REGION Network 4: First Cylinder No-3
   RUNG wire#powerrail
      Contact( "AlwaysTRUE" )
      { S7_Templates := "SrcType := Int" } Add(in1 := #Add_Cylinder[1], in2 := #Add_Cylinder[2], in3 := #Add_Cylinder[3], out => #Temp3)
      { S7_Templates := "SrcType := Int" } Sub(in1 := 3, in2 := #Temp3, out => #Temp_3)
      { S7_Templates := "value_type := Int" } SEL(g := wire#w1, in0 := #Temp_3, in1 := 3, out => #Temp_31)
      { S7_Templates := "value_type := Int" } SEL(g := wire#w2, in0 := #Temp_31, in1 := 0, out => #"First_Cylinder[3]")
   END_RUNG
   RUNG wire#powerrail
      Contact( "AlwaysTRUE" )
      Contact( #Enable_Cylinder[3] )
      Contact( #Enable_Cylinder[2] )
      Contact( #Enable_Cylinder[1] )
   END_RUNG wire#w1
   RUNG wire#powerrail
      I_Contact( #Enable_Cylinder[3] )
   END_RUNG wire#w2
   // the same network as SCL:
   // ENO of a box is taken as its EN; it also drops when the box reports an error
   IF "AlwaysTRUE" THEN
       #Temp3 := #Add_Cylinder[1] + #Add_Cylinder[2] + #Add_Cylinder[3];
       #Temp_3 := 3 - #Temp3;
       #Temp_31 := SEL(G := "AlwaysTRUE" AND #Enable_Cylinder[3] AND #Enable_Cylinder[2] AND #Enable_Cylinder[1], IN0 := #Temp_3, IN1 := 3);
       #"First_Cylinder[3]" := SEL(G := NOT #Enable_Cylinder[3], IN0 := #Temp_31, IN1 := 0);
   END_IF;
END_REGION

REGION Network 5: First Cylinder No-4
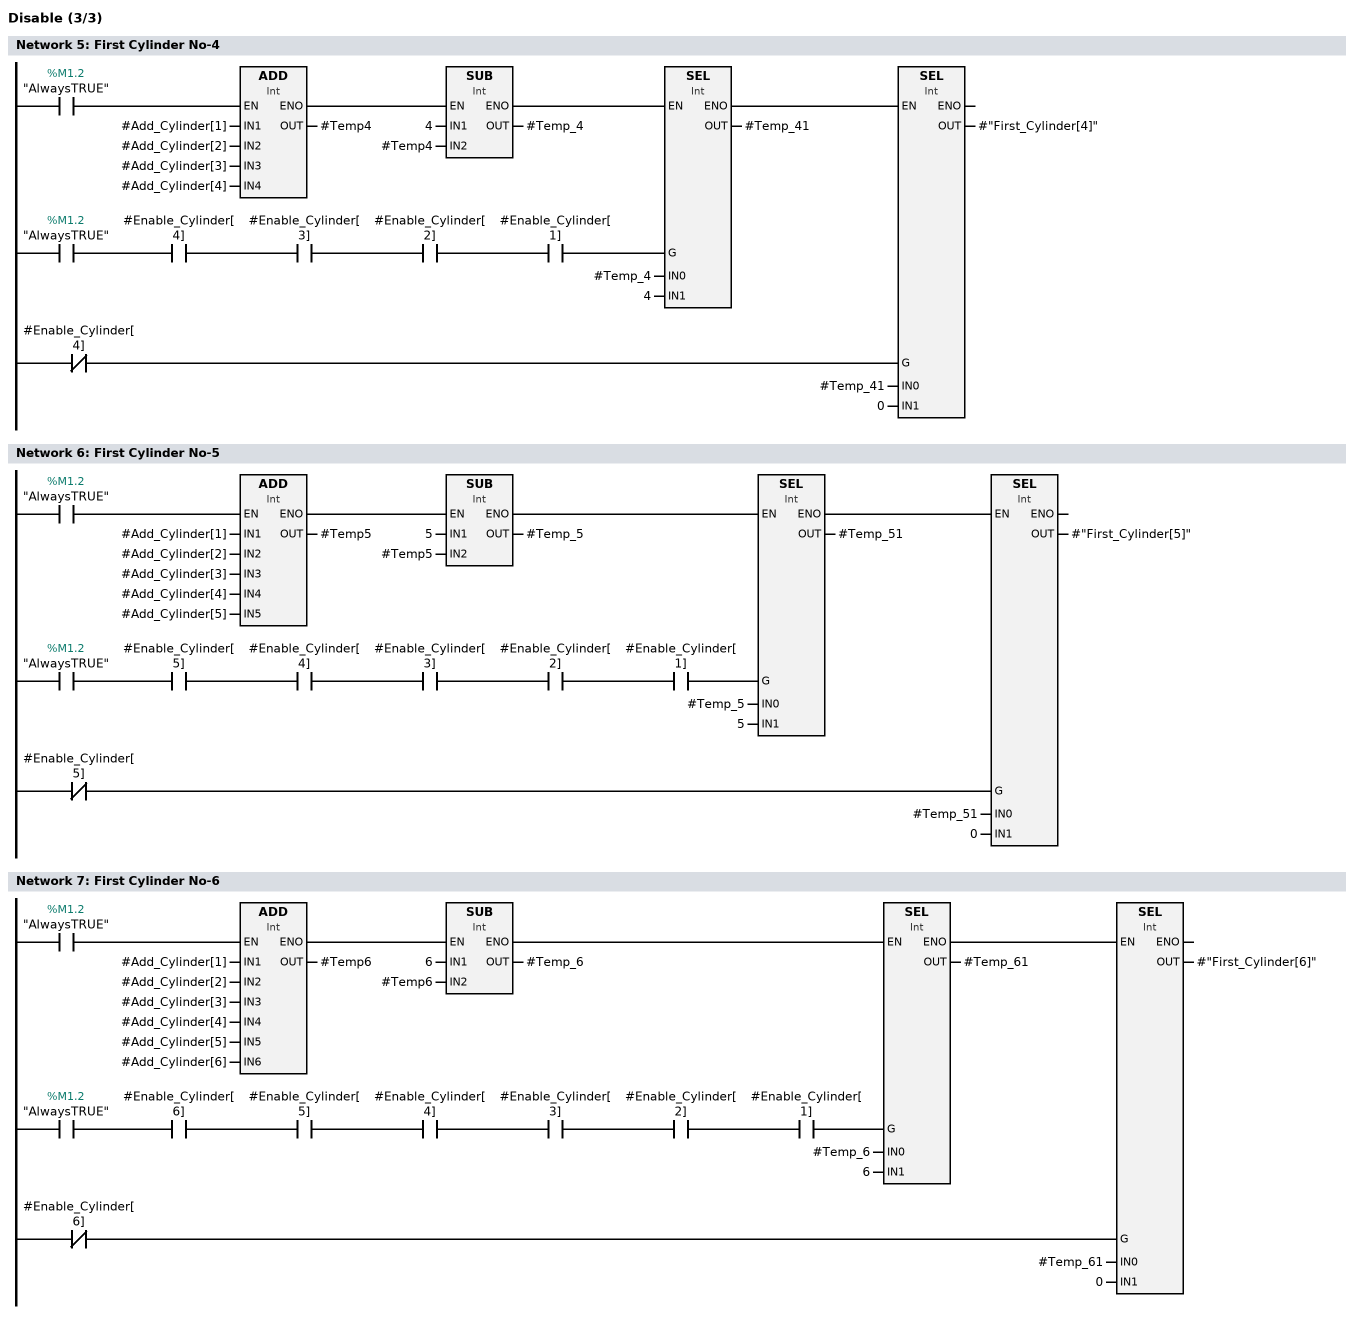
   RUNG wire#powerrail
      Contact( "AlwaysTRUE" )
      { S7_Templates := "SrcType := Int" } Add(in1 := #Add_Cylinder[1], in2 := #Add_Cylinder[2], in3 := #Add_Cylinder[3], in4 := #Add_Cylinder[4], out => #Temp4)
      { S7_Templates := "SrcType := Int" } Sub(in1 := 4, in2 := #Temp4, out => #Temp_4)
      { S7_Templates := "value_type := Int" } SEL(g := wire#w1, in0 := #Temp_4, in1 := 4, out => #Temp_41)
      { S7_Templates := "value_type := Int" } SEL(g := wire#w2, in0 := #Temp_41, in1 := 0, out => #"First_Cylinder[4]")
   END_RUNG
   RUNG wire#powerrail
      Contact( "AlwaysTRUE" )
      Contact( #Enable_Cylinder[4] )
      Contact( #Enable_Cylinder[3] )
      Contact( #Enable_Cylinder[2] )
      Contact( #Enable_Cylinder[1] )
   END_RUNG wire#w1
   RUNG wire#powerrail
      I_Contact( #Enable_Cylinder[4] )
   END_RUNG wire#w2
   // the same network as SCL:
   // ENO of a box is taken as its EN; it also drops when the box reports an error
   IF "AlwaysTRUE" THEN
       #Temp4 := #Add_Cylinder[1] + #Add_Cylinder[2] + #Add_Cylinder[3] + #Add_Cylinder[4];
       #Temp_4 := 4 - #Temp4;
       #Temp_41 := SEL(G := "AlwaysTRUE" AND #Enable_Cylinder[4] AND #Enable_Cylinder[3] AND #Enable_Cylinder[2] AND #Enable_Cylinder[1], IN0 := #Temp_4, IN1 := 4);
       #"First_Cylinder[4]" := SEL(G := NOT #Enable_Cylinder[4], IN0 := #Temp_41, IN1 := 0);
   END_IF;
END_REGION

REGION Network 6: First Cylinder No-5
   RUNG wire#powerrail
      Contact( "AlwaysTRUE" )
      { S7_Templates := "SrcType := Int" } Add(in1 := #Add_Cylinder[1], in2 := #Add_Cylinder[2], in3 := #Add_Cylinder[3], in4 := #Add_Cylinder[4], in5 := #Add_Cylinder[5], out => #Temp5)
      { S7_Templates := "SrcType := Int" } Sub(in1 := 5, in2 := #Temp5, out => #Temp_5)
      { S7_Templates := "value_type := Int" } SEL(g := wire#w1, in0 := #Temp_5, in1 := 5, out => #Temp_51)
      { S7_Templates := "value_type := Int" } SEL(g := wire#w2, in0 := #Temp_51, in1 := 0, out => #"First_Cylinder[5]")
   END_RUNG
   RUNG wire#powerrail
      Contact( "AlwaysTRUE" )
      Contact( #Enable_Cylinder[5] )
      Contact( #Enable_Cylinder[4] )
      Contact( #Enable_Cylinder[3] )
      Contact( #Enable_Cylinder[2] )
      Contact( #Enable_Cylinder[1] )
   END_RUNG wire#w1
   RUNG wire#powerrail
      I_Contact( #Enable_Cylinder[5] )
   END_RUNG wire#w2
   // the same network as SCL:
   // ENO of a box is taken as its EN; it also drops when the box reports an error
   IF "AlwaysTRUE" THEN
       #Temp5 := #Add_Cylinder[1] + #Add_Cylinder[2] + #Add_Cylinder[3] + #Add_Cylinder[4] + #Add_Cylinder[5];
       #Temp_5 := 5 - #Temp5;
       #Temp_51 := SEL(G := "AlwaysTRUE" AND #Enable_Cylinder[5] AND #Enable_Cylinder[4] AND #Enable_Cylinder[3] AND #Enable_Cylinder[2] AND #Enable_Cylinder[1], IN0 := #Temp_5, IN1 := 5);
       #"First_Cylinder[5]" := SEL(G := NOT #Enable_Cylinder[5], IN0 := #Temp_51, IN1 := 0);
   END_IF;
END_REGION

REGION Network 7: First Cylinder No-6
   RUNG wire#powerrail
      Contact( "AlwaysTRUE" )
      { S7_Templates := "SrcType := Int" } Add(in1 := #Add_Cylinder[1], in2 := #Add_Cylinder[2], in3 := #Add_Cylinder[3], in4 := #Add_Cylinder[4], in5 := #Add_Cylinder[5], in6 := #Add_Cylinder[6], out => #Temp6)
      { S7_Templates := "SrcType := Int" } Sub(in1 := 6, in2 := #Temp6, out => #Temp_6)
      { S7_Templates := "value_type := Int" } SEL(g := wire#w1, in0 := #Temp_6, in1 := 6, out => #Temp_61)
      { S7_Templates := "value_type := Int" } SEL(g := wire#w2, in0 := #Temp_61, in1 := 0, out => #"First_Cylinder[6]")
   END_RUNG
   RUNG wire#powerrail
      Contact( "AlwaysTRUE" )
      Contact( #Enable_Cylinder[6] )
      Contact( #Enable_Cylinder[5] )
      Contact( #Enable_Cylinder[4] )
      Contact( #Enable_Cylinder[3] )
      Contact( #Enable_Cylinder[2] )
      Contact( #Enable_Cylinder[1] )
   END_RUNG wire#w1
   RUNG wire#powerrail
      I_Contact( #Enable_Cylinder[6] )
   END_RUNG wire#w2
   // the same network as SCL:
   // ENO of a box is taken as its EN; it also drops when the box reports an error
   IF "AlwaysTRUE" THEN
       #Temp6 := #Add_Cylinder[1] + #Add_Cylinder[2] + #Add_Cylinder[3] + #Add_Cylinder[4] + #Add_Cylinder[5] + #Add_Cylinder[6];
       #Temp_6 := 6 - #Temp6;
       #Temp_61 := SEL(G := "AlwaysTRUE" AND #Enable_Cylinder[6] AND #Enable_Cylinder[5] AND #Enable_Cylinder[4] AND #Enable_Cylinder[3] AND #Enable_Cylinder[2] AND #Enable_Cylinder[1], IN0 := #Temp_6, IN1 := 6);
       #"First_Cylinder[6]" := SEL(G := NOT #Enable_Cylinder[6], IN0 := #Temp_61, IN1 := 0);
   END_IF;
END_REGION
END_FUNCTION_BLOCK

FUNCTION_BLOCK "LPG_FILLING_FB"   // FB101, LAD
TITLE = Fiiling Operation FB
{ S7_Optimized_Access := 'TRUE' }
VERSION : 0.1
// stored: AutoNumber false, IsIECCheckEnabled false, IsRetainMemResEnabled false, MemoryReserve 100, SetENOAutomatically false, UDAEnableTagReadback false
   VAR_INPUT
      INxCylinder_In_Pos : Bool;   // Cylinder In Position
      INxAuto_Start_Seq : Bool;   // Start Filling Sequence
      INxMan_Start_Seq : Bool;
      INxStop_Sequence : Bool;   // Stop Filling Sequence
      INtStart_TImeout_Time : DInt;   // Start Timeout Time in Sec
      INxReset_Sequence : Bool;   // Reset Sequence
      INxCylinder_Type : Int;
      INrTare_Entry_SP : Real;
      ALL_FILL_DONE : Bool;
      DOWN_CONVEYOR : Bool;
   END_VAR
   VAR_OUTPUT
      OutuFilled_Data : Array[1..3] of Real;
      OutxDomestic_Cylinder : Bool;
      OutxCommercial_Cylinder : Bool;
      OutxStart_Timeout : Bool;
      OutxTare_Entry_Error : Bool;   // Coil 27
      Outx_Filling_Error : Bool;
      Outx_Tare_Value_Error : Bool;
      Cycle_Started : Bool;
      OutiStep_No : Int;
      OUTxFilling_Done : Bool;
      Gross_Weight : Real;
      Net_Wieght : Real;
      Tare_Weight : Real;
   END_VAR
   VAR_IN_OUT
      Modbus_Master_DB : "MOD_MASTER_DATA";
   END_VAR
   VAR
      TRIG : Array[1..25] of Bool;
      STEP_NO : Int;
      Step_Timer { S7_SetPoint := 'True'} : Array[1..15] of IEC_TIMER;
      Domestic_Cylinder { S7_SetPoint := 'True'} : Bool;
      Commercial_Cylinder : Bool;
      Cyl_Done { S7_SetPoint := 'True'} : TOF_TIME;
      Tare_Enrty_Extn { S7_SetPoint := 'True'} : TOF_TIME;
      Start_Timeout_Err { S7_SetPoint := 'True'} : TON_TIME;
      Tare_Entry_Timer { S7_SetPoint := 'True'} : TON_TIME;
      Filled_Gross : Real;
      Filled_Net : Real;
      Punched_Tare : Real;
      Test_Seq : Int;
      Filling_Done : Bool;
      IEC_Timer_0_Instance { S7_SetPoint := 'True'} : TOF_TIME;
      Gross { S7_SetPoint := 'True'} : Real;
      gross_diff : Real;
      pass : Bool;
   END_VAR
   VAR_TEMP
      Tare_Weight_Mul : Real;
      Tare_Enter_Time : DInt;
      Stt_TImeout_Time : DInt;
      Tare_Entry_Time : DInt;
      Tare_SP_Weigher : Int;
      Filled_Gross_Mul : Int;
      Filled_Net_Mul : Int;
      Filled_Tare_Mul : Int;
      "final wieght" : Real;
      final_weight_1 : Real;
   END_VAR
   // Tare_Enrty_Extn.PT := T#1s;
   VAR_TEMP   // added for the SCL form of the ladder/FBD networks
      _w1 : Bool;
      _w2 : Bool;
      _w3 : Bool;
   END_VAR
BEGIN

REGION Network 1: Empty Network
END_REGION

REGION Network 2: Input Mapping
END_REGION

REGION Network 3: Cylinder Selection ( Domestic / Commercial )
   // We have to receive from FIFO Entry-
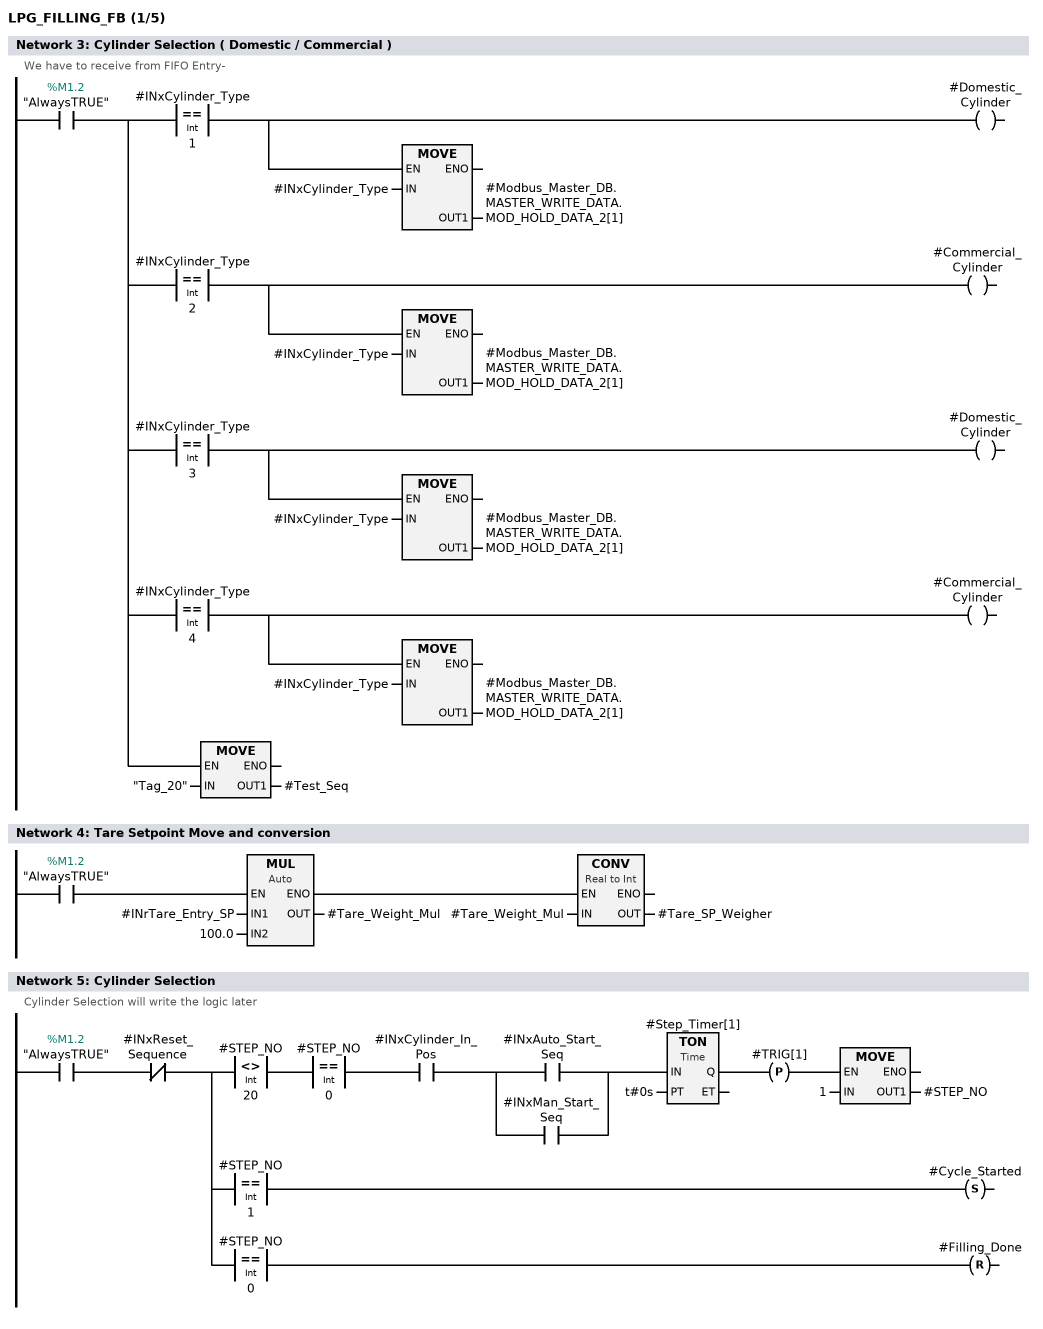
   RUNG wire#powerrail
      Contact( "AlwaysTRUE" )
      wire#w1
      { S7_Templates := "SrcType := Int" } EQ_Contact(in1 := #INxCylinder_Type, in2 := 1)
      wire#w2
      Coil( #Domestic_Cylinder )
   END_RUNG
   RUNG wire#w2
      Move(in := #INxCylinder_Type, out1 => #Modbus_Master_DB.MASTER_WRITE_DATA.MOD_HOLD_DATA_2[1])
   END_RUNG
   RUNG wire#w1
      { S7_Templates := "SrcType := Int" } EQ_Contact(in1 := #INxCylinder_Type, in2 := 2)
      wire#w3
      Coil( #Commercial_Cylinder )
   END_RUNG
   RUNG wire#w3
      Move(in := #INxCylinder_Type, out1 => #Modbus_Master_DB.MASTER_WRITE_DATA.MOD_HOLD_DATA_2[1])
   END_RUNG
   RUNG wire#w1
      { S7_Templates := "SrcType := Int" } EQ_Contact(in1 := #INxCylinder_Type, in2 := 3)
      wire#w4
      Coil( #Domestic_Cylinder )
   END_RUNG
   RUNG wire#w4
      Move(in := #INxCylinder_Type, out1 => #Modbus_Master_DB.MASTER_WRITE_DATA.MOD_HOLD_DATA_2[1])
   END_RUNG
   RUNG wire#w1
      { S7_Templates := "SrcType := Int" } EQ_Contact(in1 := #INxCylinder_Type, in2 := 4)
      wire#w5
      Coil( #Commercial_Cylinder )
   END_RUNG
   RUNG wire#w5
      Move(in := #INxCylinder_Type, out1 => #Modbus_Master_DB.MASTER_WRITE_DATA.MOD_HOLD_DATA_2[1])
   END_RUNG
   RUNG wire#w1
      Move(in := "Tag_20", out1 => #Test_Seq)
   END_RUNG
   // the same network as SCL:
   #Domestic_Cylinder := "AlwaysTRUE" AND (#INxCylinder_Type = 1);
   IF #Domestic_Cylinder THEN
       #Modbus_Master_DB.MASTER_WRITE_DATA.MOD_HOLD_DATA_2[1] := #INxCylinder_Type;
   END_IF;
   #Commercial_Cylinder := "AlwaysTRUE" AND (#INxCylinder_Type = 2);
   IF #Commercial_Cylinder THEN
       #Modbus_Master_DB.MASTER_WRITE_DATA.MOD_HOLD_DATA_2[1] := #INxCylinder_Type;
   END_IF;
   #Domestic_Cylinder := "AlwaysTRUE" AND (#INxCylinder_Type = 3);
   IF #Domestic_Cylinder THEN
       #Modbus_Master_DB.MASTER_WRITE_DATA.MOD_HOLD_DATA_2[1] := #INxCylinder_Type;
   END_IF;
   #Commercial_Cylinder := "AlwaysTRUE" AND (#INxCylinder_Type = 4);
   IF #Commercial_Cylinder THEN
       #Modbus_Master_DB.MASTER_WRITE_DATA.MOD_HOLD_DATA_2[1] := #INxCylinder_Type;
   END_IF;
   IF "AlwaysTRUE" THEN #Test_Seq := "Tag_20"; END_IF;
END_REGION

REGION Network 4: Tare Setpoint Move and conversion
   RUNG wire#powerrail
      Contact( "AlwaysTRUE" )
      Mul(in1 := #INrTare_Entry_SP, in2 := 100.0, out => #Tare_Weight_Mul)
      { S7_Templates := "[SrcType := Real, DestType := Int]" } Convert(in := #Tare_Weight_Mul, out => #Tare_SP_Weigher)
   END_RUNG
   // the same network as SCL:
   IF "AlwaysTRUE" THEN
       #Tare_Weight_Mul := #INrTare_Entry_SP * 100.0;
       #Tare_SP_Weigher := REAL_TO_INT(#Tare_Weight_Mul);
   END_IF;
END_REGION

REGION Network 5: Cylinder Selection
   // Cylinder Selection will write the logic later
   RUNG wire#powerrail
      Contact( "AlwaysTRUE" )
      I_Contact( #INxReset_Sequence )
      wire#w1
      { S7_Templates := "SrcType := Int" } NE_Contact(in1 := #STEP_NO, in2 := 20)
      { S7_Templates := "SrcType := Int" } EQ_Contact(in1 := #STEP_NO, in2 := 0)
      Contact( #INxCylinder_In_Pos )
      wire#w2
      Contact( #INxAuto_Start_Seq )
      wire#w3
      { S7_Templates := "time_type := Time" } #Step_Timer[1].TON(pt := t#0s, et =>)
      P_Trig( #TRIG[1] )
      Move(in := 1, out1 => #STEP_NO)
   END_RUNG
   RUNG wire#w2
      Contact( #INxMan_Start_Seq )
   END_RUNG wire#w3
   RUNG wire#w1
      { S7_Templates := "SrcType := Int" } EQ_Contact(in1 := #STEP_NO, in2 := 1)
      S_Coil( #Cycle_Started )
   END_RUNG
   RUNG wire#w1
      { S7_Templates := "SrcType := Int" } EQ_Contact(in1 := #STEP_NO, in2 := 0)
      R_Coil( #Filling_Done )
   END_RUNG
   // the same network as SCL:
   #_w1 := "AlwaysTRUE" AND NOT #INxReset_Sequence;
   #Step_Timer[1].TON(IN := #_w1 AND (#STEP_NO <> 20) AND (#STEP_NO = 0) AND #INxCylinder_In_Pos AND (#INxAuto_Start_Seq OR #INxMan_Start_Seq),
                      PT := t#0s);
   #_w2 := #Step_Timer[1].Q AND NOT #TRIG[1];   // rising edge
   #TRIG[1] := #Step_Timer[1].Q;
   IF #_w2 THEN #STEP_NO := 1; END_IF;
   IF #_w1 AND (#STEP_NO = 1) THEN #Cycle_Started := TRUE; END_IF;
   IF #_w1 AND (#STEP_NO = 0) THEN #Filling_Done := FALSE; END_IF;
END_REGION

REGION Network 6: Check the Cylinder In Position
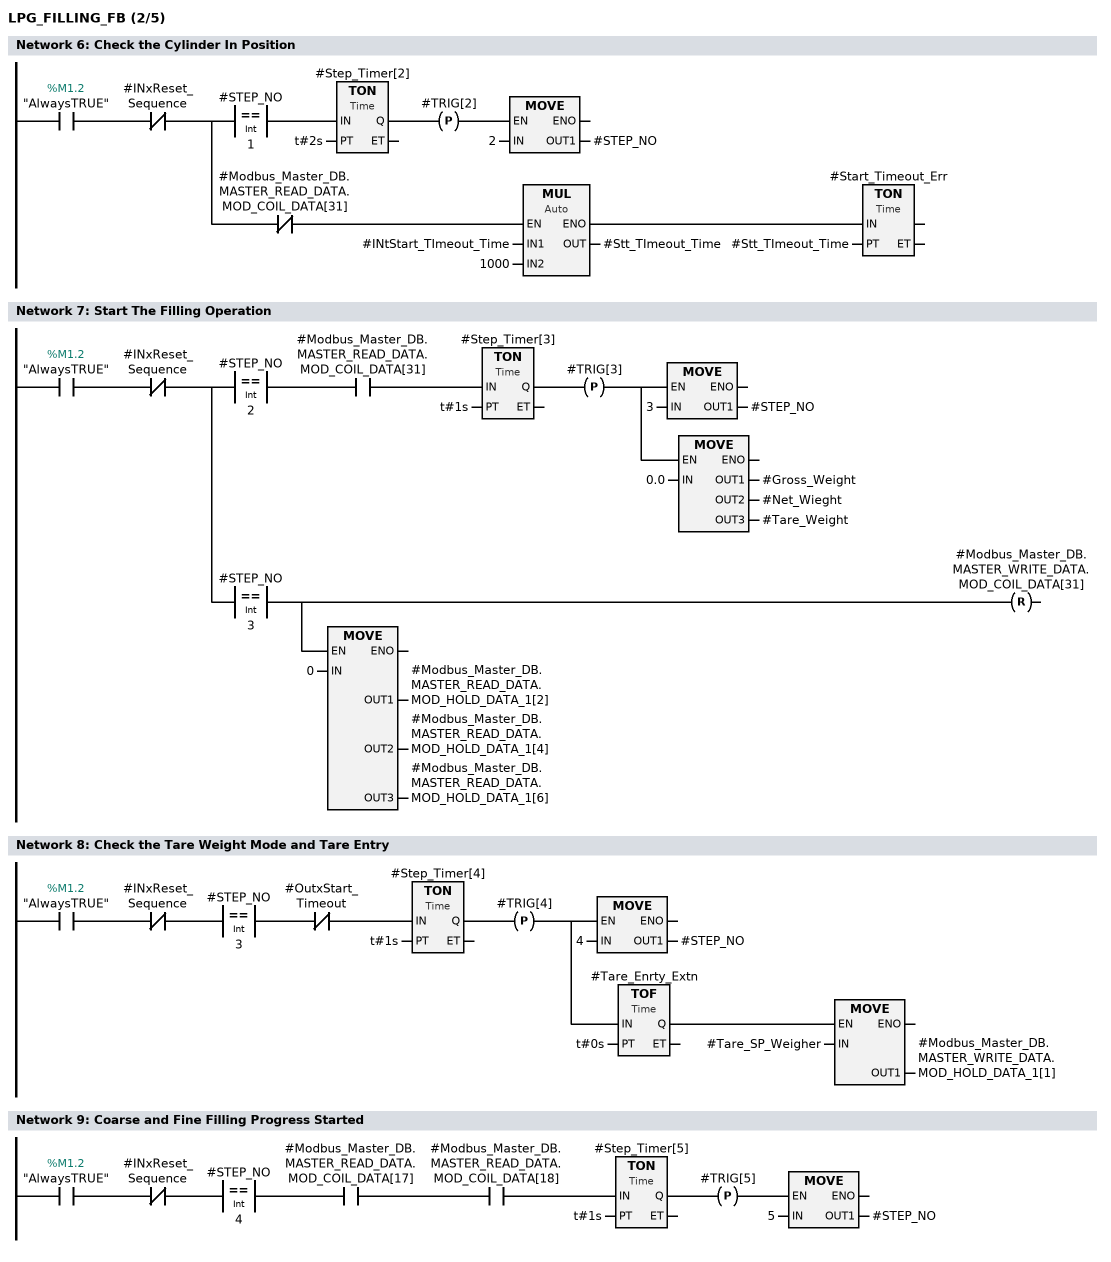
   RUNG wire#powerrail
      Contact( "AlwaysTRUE" )
      I_Contact( #INxReset_Sequence )
      wire#w1
      { S7_Templates := "SrcType := Int" } EQ_Contact(in1 := #STEP_NO, in2 := 1)
      { S7_Templates := "time_type := Time" } #Step_Timer[2].TON(pt := t#2s, et =>)
      P_Trig( #TRIG[2] )
      Move(in := 2, out1 => #STEP_NO)
   END_RUNG
   RUNG wire#w1
      I_Contact( #Modbus_Master_DB.MASTER_READ_DATA.MOD_COIL_DATA[31] )
      Mul(in1 := #INtStart_TImeout_Time, in2 := 1000, out => #Stt_TImeout_Time)
      { S7_Templates := "time_type := Time" } #Start_Timeout_Err.TON(pt := #Stt_TImeout_Time, et =>)
   END_RUNG
   // the same network as SCL:
   #_w1 := "AlwaysTRUE" AND NOT #INxReset_Sequence;
   #Step_Timer[2].TON(IN := #_w1 AND (#STEP_NO = 1), PT := t#2s);
   #_w2 := #Step_Timer[2].Q AND NOT #TRIG[2];   // rising edge
   #TRIG[2] := #Step_Timer[2].Q;
   IF #_w2 THEN #STEP_NO := 2; END_IF;
   #_w3 := #_w1 AND NOT #Modbus_Master_DB.MASTER_READ_DATA.MOD_COIL_DATA[31];
   IF #_w3 THEN #Stt_TImeout_Time := #INtStart_TImeout_Time * 1000; END_IF;
   #Start_Timeout_Err(IN := #_w3, PT := #Stt_TImeout_Time);   // TON
END_REGION

REGION Network 7: Start The Filling Operation
   RUNG wire#powerrail
      Contact( "AlwaysTRUE" )
      I_Contact( #INxReset_Sequence )
      wire#w1
      { S7_Templates := "SrcType := Int" } EQ_Contact(in1 := #STEP_NO, in2 := 2)
      Contact( #Modbus_Master_DB.MASTER_READ_DATA.MOD_COIL_DATA[31] )
      { S7_Templates := "time_type := Time" } #Step_Timer[3].TON(pt := t#1s, et =>)
      P_Trig( #TRIG[3] )
      wire#w2
      Move(in := 3, out1 => #STEP_NO)
   END_RUNG
   RUNG wire#w2
      Move(in := 0.0, out1 => #Gross_Weight, out2 => #Net_Wieght, out3 => #Tare_Weight)
   END_RUNG
   RUNG wire#w1
      { S7_Templates := "SrcType := Int" } EQ_Contact(in1 := #STEP_NO, in2 := 3)
      wire#w3
      R_Coil( #Modbus_Master_DB.MASTER_WRITE_DATA.MOD_COIL_DATA[31] )
   END_RUNG
   RUNG wire#w3
      Move(in := 0, out1 => #Modbus_Master_DB.MASTER_READ_DATA.MOD_HOLD_DATA_1[2], out2 => #Modbus_Master_DB.MASTER_READ_DATA.MOD_HOLD_DATA_1[4], out3 => #Modbus_Master_DB.MASTER_READ_DATA.MOD_HOLD_DATA_1[6])
   END_RUNG
   // the same network as SCL:
   #_w1 := "AlwaysTRUE" AND NOT #INxReset_Sequence;
   #Step_Timer[3].TON(IN := #_w1 AND (#STEP_NO = 2) AND #Modbus_Master_DB.MASTER_READ_DATA.MOD_COIL_DATA[31],
                      PT := t#1s);
   #_w2 := #Step_Timer[3].Q AND NOT #TRIG[3];   // rising edge
   #TRIG[3] := #Step_Timer[3].Q;
   IF #_w2 THEN
       #STEP_NO := 3;
       #Gross_Weight := 0.0;
       #Net_Wieght := 0.0;
       #Tare_Weight := 0.0;
   END_IF;
   IF #_w1 AND (#STEP_NO = 3) THEN
       #Modbus_Master_DB.MASTER_WRITE_DATA.MOD_COIL_DATA[31] := FALSE;
       #Modbus_Master_DB.MASTER_READ_DATA.MOD_HOLD_DATA_1[2] := 0;
       #Modbus_Master_DB.MASTER_READ_DATA.MOD_HOLD_DATA_1[4] := 0;
       #Modbus_Master_DB.MASTER_READ_DATA.MOD_HOLD_DATA_1[6] := 0;
   END_IF;
END_REGION

REGION Network 8: Check the Tare Weight Mode and Tare Entry
   RUNG wire#powerrail
      Contact( "AlwaysTRUE" )
      I_Contact( #INxReset_Sequence )
      { S7_Templates := "SrcType := Int" } EQ_Contact(in1 := #STEP_NO, in2 := 3)
      I_Contact( #OutxStart_Timeout )
      { S7_Templates := "time_type := Time" } #Step_Timer[4].TON(pt := t#1s, et =>)
      P_Trig( #TRIG[4] )
      wire#w1
      Move(in := 4, out1 => #STEP_NO)
   END_RUNG
   RUNG wire#w1
      { S7_Templates := "time_type := Time" } #Tare_Enrty_Extn.TOF(pt := t#0s, et =>)
      Move(in := #Tare_SP_Weigher, out1 => #Modbus_Master_DB.MASTER_WRITE_DATA.MOD_HOLD_DATA_1[1])
   END_RUNG
   // the same network as SCL:
   #Step_Timer[4].TON(IN := "AlwaysTRUE" AND NOT #INxReset_Sequence AND (#STEP_NO = 3) AND NOT #OutxStart_Timeout,
                      PT := t#1s);
   #_w1 := #Step_Timer[4].Q AND NOT #TRIG[4];   // rising edge
   #TRIG[4] := #Step_Timer[4].Q;
   IF #_w1 THEN #STEP_NO := 4; END_IF;
   #Tare_Enrty_Extn(IN := #_w1, PT := t#0s);   // TOF
   IF #Tare_Enrty_Extn.Q THEN
       #Modbus_Master_DB.MASTER_WRITE_DATA.MOD_HOLD_DATA_1[1] := #Tare_SP_Weigher;
   END_IF;
END_REGION

REGION Network 9: Coarse and Fine Filling Progress Started
   RUNG wire#powerrail
      Contact( "AlwaysTRUE" )
      I_Contact( #INxReset_Sequence )
      { S7_Templates := "SrcType := Int" } EQ_Contact(in1 := #STEP_NO, in2 := 4)
      Contact( #Modbus_Master_DB.MASTER_READ_DATA.MOD_COIL_DATA[17] )
      Contact( #Modbus_Master_DB.MASTER_READ_DATA.MOD_COIL_DATA[18] )
      { S7_Templates := "time_type := Time" } #Step_Timer[5].TON(pt := t#1s, et =>)
      P_Trig( #TRIG[5] )
      Move(in := 5, out1 => #STEP_NO)
   END_RUNG
   // the same network as SCL:
   #Step_Timer[5].TON(IN := "AlwaysTRUE" AND NOT #INxReset_Sequence AND (#STEP_NO = 4) AND #Modbus_Master_DB.MASTER_READ_DATA.MOD_COIL_DATA[17] AND #Modbus_Master_DB.MASTER_READ_DATA.MOD_COIL_DATA[18],
                      PT := t#1s);
   #_w1 := #Step_Timer[5].Q AND NOT #TRIG[5];   // rising edge
   #TRIG[5] := #Step_Timer[5].Q;
   IF #_w1 THEN #STEP_NO := 5; END_IF;
END_REGION

REGION Network 10: Coarse Filling Completed
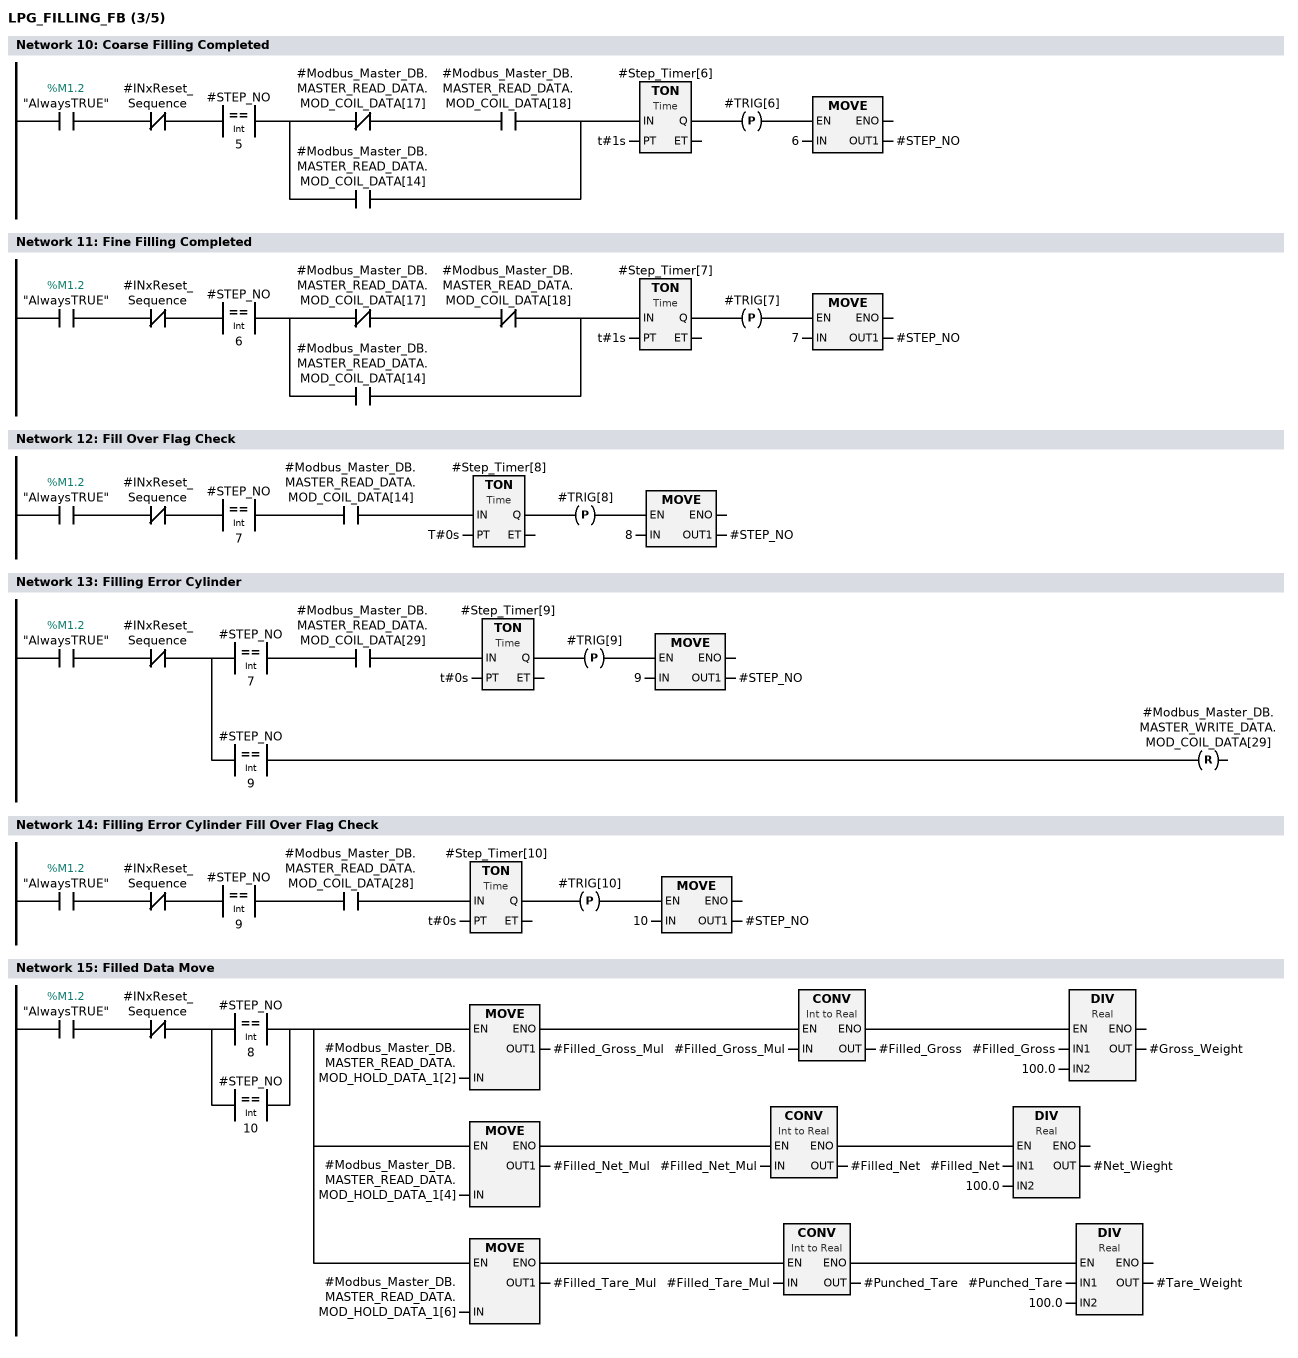
   RUNG wire#powerrail
      Contact( "AlwaysTRUE" )
      I_Contact( #INxReset_Sequence )
      { S7_Templates := "SrcType := Int" } EQ_Contact(in1 := #STEP_NO, in2 := 5)
      wire#w1
      I_Contact( #Modbus_Master_DB.MASTER_READ_DATA.MOD_COIL_DATA[17] )
      Contact( #Modbus_Master_DB.MASTER_READ_DATA.MOD_COIL_DATA[18] )
      wire#w2
      { S7_Templates := "time_type := Time" } #Step_Timer[6].TON(pt := t#1s, et =>)
      P_Trig( #TRIG[6] )
      Move(in := 6, out1 => #STEP_NO)
   END_RUNG
   RUNG wire#w1
      Contact( #Modbus_Master_DB.MASTER_READ_DATA.MOD_COIL_DATA[14] )
   END_RUNG wire#w2
   // the same network as SCL:
   #Step_Timer[6].TON(IN := "AlwaysTRUE" AND NOT #INxReset_Sequence AND (#STEP_NO = 5) AND ((NOT #Modbus_Master_DB.MASTER_READ_DATA.MOD_COIL_DATA[17] AND #Modbus_Master_DB.MASTER_READ_DATA.MOD_COIL_DATA[18]) OR #Modbus_Master_DB.MASTER_READ_DATA.MOD_COIL_DATA[14]),
                      PT := t#1s);
   #_w1 := #Step_Timer[6].Q AND NOT #TRIG[6];   // rising edge
   #TRIG[6] := #Step_Timer[6].Q;
   IF #_w1 THEN #STEP_NO := 6; END_IF;
END_REGION

REGION Network 11: Fine Filling Completed
   RUNG wire#powerrail
      Contact( "AlwaysTRUE" )
      I_Contact( #INxReset_Sequence )
      { S7_Templates := "SrcType := Int" } EQ_Contact(in1 := #STEP_NO, in2 := 6)
      wire#w1
      I_Contact( #Modbus_Master_DB.MASTER_READ_DATA.MOD_COIL_DATA[17] )
      I_Contact( #Modbus_Master_DB.MASTER_READ_DATA.MOD_COIL_DATA[18] )
      wire#w2
      { S7_Templates := "time_type := Time" } #Step_Timer[7].TON(pt := t#1s, et =>)
      P_Trig( #TRIG[7] )
      Move(in := 7, out1 => #STEP_NO)
   END_RUNG
   RUNG wire#w1
      Contact( #Modbus_Master_DB.MASTER_READ_DATA.MOD_COIL_DATA[14] )
   END_RUNG wire#w2
   // the same network as SCL:
   #Step_Timer[7].TON(IN := "AlwaysTRUE" AND NOT #INxReset_Sequence AND (#STEP_NO = 6) AND ((NOT #Modbus_Master_DB.MASTER_READ_DATA.MOD_COIL_DATA[17] AND NOT #Modbus_Master_DB.MASTER_READ_DATA.MOD_COIL_DATA[18]) OR #Modbus_Master_DB.MASTER_READ_DATA.MOD_COIL_DATA[14]),
                      PT := t#1s);
   #_w1 := #Step_Timer[7].Q AND NOT #TRIG[7];   // rising edge
   #TRIG[7] := #Step_Timer[7].Q;
   IF #_w1 THEN #STEP_NO := 7; END_IF;
END_REGION

REGION Network 12: Fill Over Flag Check
   RUNG wire#powerrail
      Contact( "AlwaysTRUE" )
      I_Contact( #INxReset_Sequence )
      { S7_Templates := "SrcType := Int" } EQ_Contact(in1 := #STEP_NO, in2 := 7)
      Contact( #Modbus_Master_DB.MASTER_READ_DATA.MOD_COIL_DATA[14] )
      { S7_Templates := "time_type := Time" } #Step_Timer[8].TON(pt := T#0s, et =>)
      P_Trig( #TRIG[8] )
      Move(in := 8, out1 => #STEP_NO)
   END_RUNG
   // the same network as SCL:
   #Step_Timer[8].TON(IN := "AlwaysTRUE" AND NOT #INxReset_Sequence AND (#STEP_NO = 7) AND #Modbus_Master_DB.MASTER_READ_DATA.MOD_COIL_DATA[14],
                      PT := T#0s);
   #_w1 := #Step_Timer[8].Q AND NOT #TRIG[8];   // rising edge
   #TRIG[8] := #Step_Timer[8].Q;
   IF #_w1 THEN #STEP_NO := 8; END_IF;
END_REGION

REGION Network 13: Filling Error Cylinder
   RUNG wire#powerrail
      Contact( "AlwaysTRUE" )
      I_Contact( #INxReset_Sequence )
      wire#w1
      { S7_Templates := "SrcType := Int" } EQ_Contact(in1 := #STEP_NO, in2 := 7)
      Contact( #Modbus_Master_DB.MASTER_READ_DATA.MOD_COIL_DATA[29] )
      { S7_Templates := "time_type := Time" } #Step_Timer[9].TON(pt := t#0s, et =>)
      P_Trig( #TRIG[9] )
      Move(in := 9, out1 => #STEP_NO)
   END_RUNG
   RUNG wire#w1
      { S7_Templates := "SrcType := Int" } EQ_Contact(in1 := #STEP_NO, in2 := 9)
      R_Coil( #Modbus_Master_DB.MASTER_WRITE_DATA.MOD_COIL_DATA[29] )
   END_RUNG
   // the same network as SCL:
   #_w1 := "AlwaysTRUE" AND NOT #INxReset_Sequence;
   #Step_Timer[9].TON(IN := #_w1 AND (#STEP_NO = 7) AND #Modbus_Master_DB.MASTER_READ_DATA.MOD_COIL_DATA[29],
                      PT := t#0s);
   #_w2 := #Step_Timer[9].Q AND NOT #TRIG[9];   // rising edge
   #TRIG[9] := #Step_Timer[9].Q;
   IF #_w2 THEN #STEP_NO := 9; END_IF;
   IF #_w1 AND (#STEP_NO = 9) THEN #Modbus_Master_DB.MASTER_WRITE_DATA.MOD_COIL_DATA[29] := FALSE; END_IF;
END_REGION

REGION Network 14: Filling Error Cylinder Fill Over Flag Check
   RUNG wire#powerrail
      Contact( "AlwaysTRUE" )
      I_Contact( #INxReset_Sequence )
      { S7_Templates := "SrcType := Int" } EQ_Contact(in1 := #STEP_NO, in2 := 9)
      Contact( #Modbus_Master_DB.MASTER_READ_DATA.MOD_COIL_DATA[28] )
      { S7_Templates := "time_type := Time" } #Step_Timer[10].TON(pt := t#0s, et =>)
      P_Trig( #TRIG[10] )
      Move(in := 10, out1 => #STEP_NO)
   END_RUNG
   // the same network as SCL:
   #Step_Timer[10].TON(IN := "AlwaysTRUE" AND NOT #INxReset_Sequence AND (#STEP_NO = 9) AND #Modbus_Master_DB.MASTER_READ_DATA.MOD_COIL_DATA[28],
                       PT := t#0s);
   #_w1 := #Step_Timer[10].Q AND NOT #TRIG[10];   // rising edge
   #TRIG[10] := #Step_Timer[10].Q;
   IF #_w1 THEN #STEP_NO := 10; END_IF;
END_REGION

REGION Network 15: Filled Data Move
   RUNG wire#powerrail
      Contact( "AlwaysTRUE" )
      I_Contact( #INxReset_Sequence )
      wire#w1
      { S7_Templates := "SrcType := Int" } EQ_Contact(in1 := #STEP_NO, in2 := 8)
      wire#w2
      Move(in := #Modbus_Master_DB.MASTER_READ_DATA.MOD_HOLD_DATA_1[2], out1 => #Filled_Gross_Mul)
      { S7_Templates := "[SrcType := Int, DestType := Real]" } Convert(in := #Filled_Gross_Mul, out => #Filled_Gross)
      { S7_Templates := "SrcType := Real" } Div(in1 := #Filled_Gross, in2 := 100.0, out => #Gross_Weight)
   END_RUNG
   RUNG wire#w1
      { S7_Templates := "SrcType := Int" } EQ_Contact(in1 := #STEP_NO, in2 := 10)
   END_RUNG wire#w2
   RUNG wire#w2
      Move(in := #Modbus_Master_DB.MASTER_READ_DATA.MOD_HOLD_DATA_1[4], out1 => #Filled_Net_Mul)
      { S7_Templates := "[SrcType := Int, DestType := Real]" } Convert(in := #Filled_Net_Mul, out => #Filled_Net)
      { S7_Templates := "SrcType := Real" } Div(in1 := #Filled_Net, in2 := 100.0, out => #Net_Wieght)
   END_RUNG
   RUNG wire#w2
      Move(in := #Modbus_Master_DB.MASTER_READ_DATA.MOD_HOLD_DATA_1[6], out1 => #Filled_Tare_Mul)
      { S7_Templates := "[SrcType := Int, DestType := Real]" } Convert(in := #Filled_Tare_Mul, out => #Punched_Tare)
      { S7_Templates := "SrcType := Real" } Div(in1 := #Punched_Tare, in2 := 100.0, out => #Tare_Weight)
   END_RUNG
   // the same network as SCL:
   IF "AlwaysTRUE" AND NOT #INxReset_Sequence AND ((#STEP_NO = 8) OR (#STEP_NO = 10)) THEN
       #Filled_Gross_Mul := #Modbus_Master_DB.MASTER_READ_DATA.MOD_HOLD_DATA_1[2];
       #Filled_Gross := INT_TO_REAL(#Filled_Gross_Mul);
       #Gross_Weight := #Filled_Gross / 100.0;
       #Filled_Net_Mul := #Modbus_Master_DB.MASTER_READ_DATA.MOD_HOLD_DATA_1[4];
       #Filled_Net := INT_TO_REAL(#Filled_Net_Mul);
       #Net_Wieght := #Filled_Net / 100.0;
       #Filled_Tare_Mul := #Modbus_Master_DB.MASTER_READ_DATA.MOD_HOLD_DATA_1[6];
       #Punched_Tare := INT_TO_REAL(#Filled_Tare_Mul);
       #Tare_Weight := #Punched_Tare / 100.0;
   END_IF;
END_REGION

REGION Network 16: Filling Operation Complete
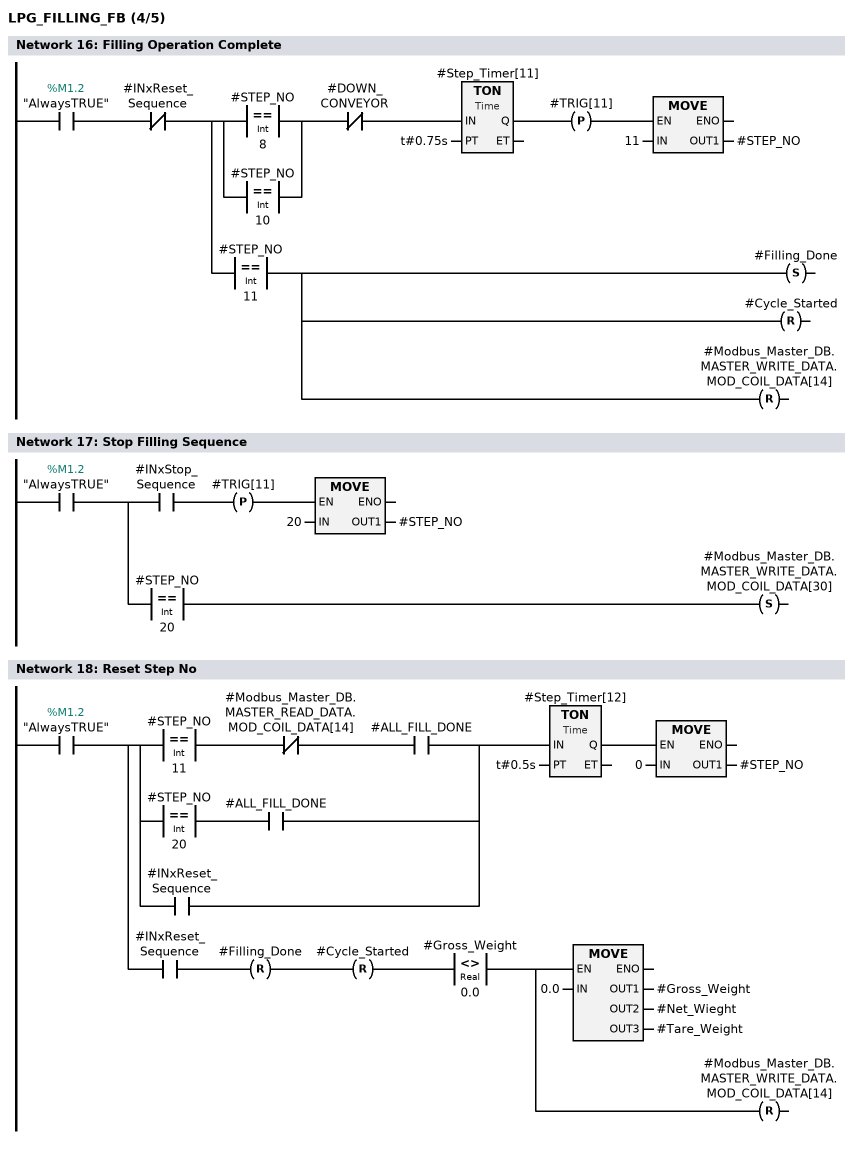
   RUNG wire#powerrail
      Contact( "AlwaysTRUE" )
      I_Contact( #INxReset_Sequence )
      wire#w1
      { S7_Templates := "SrcType := Int" } EQ_Contact(in1 := #STEP_NO, in2 := 8)
      wire#w2
      I_Contact( #DOWN_CONVEYOR )
      { S7_Templates := "time_type := Time" } #Step_Timer[11].TON(pt := t#0.75s, et =>)
      P_Trig( #TRIG[11] )
      Move(in := 11, out1 => #STEP_NO)
   END_RUNG
   RUNG wire#w1
      { S7_Templates := "SrcType := Int" } EQ_Contact(in1 := #STEP_NO, in2 := 10)
   END_RUNG wire#w2
   RUNG wire#w1
      { S7_Templates := "SrcType := Int" } EQ_Contact(in1 := #STEP_NO, in2 := 11)
      wire#w3
      S_Coil( #Filling_Done )
   END_RUNG
   RUNG wire#w3
      R_Coil( #Cycle_Started )
   END_RUNG
   RUNG wire#w3
      R_Coil( #Modbus_Master_DB.MASTER_WRITE_DATA.MOD_COIL_DATA[14] )
   END_RUNG
   // the same network as SCL:
   #_w1 := "AlwaysTRUE" AND NOT #INxReset_Sequence;
   #Step_Timer[11].TON(IN := #_w1 AND ((#STEP_NO = 8) OR (#STEP_NO = 10)) AND NOT #DOWN_CONVEYOR, PT := t#0.75s);
   #_w2 := #Step_Timer[11].Q AND NOT #TRIG[11];   // rising edge
   #TRIG[11] := #Step_Timer[11].Q;
   IF #_w2 THEN #STEP_NO := 11; END_IF;
   IF #_w1 AND (#STEP_NO = 11) THEN
       #Filling_Done := TRUE;
       #Cycle_Started := FALSE;
       #Modbus_Master_DB.MASTER_WRITE_DATA.MOD_COIL_DATA[14] := FALSE;
   END_IF;
END_REGION

REGION Network 17: Stop Filling Sequence
   RUNG wire#powerrail
      Contact( "AlwaysTRUE" )
      wire#w1
      Contact( #INxStop_Sequence )
      P_Trig( #TRIG[11] )
      Move(in := 20, out1 => #STEP_NO)
   END_RUNG
   RUNG wire#w1
      { S7_Templates := "SrcType := Int" } EQ_Contact(in1 := #STEP_NO, in2 := 20)
      S_Coil( #Modbus_Master_DB.MASTER_WRITE_DATA.MOD_COIL_DATA[30] )
   END_RUNG
   // the same network as SCL:
   #_w1 := "AlwaysTRUE" AND #INxStop_Sequence;
   #_w2 := #_w1 AND NOT #TRIG[11];   // rising edge
   #TRIG[11] := #_w1;
   IF #_w2 THEN #STEP_NO := 20; END_IF;
   IF "AlwaysTRUE" AND (#STEP_NO = 20) THEN
       #Modbus_Master_DB.MASTER_WRITE_DATA.MOD_COIL_DATA[30] := TRUE;
   END_IF;
END_REGION

REGION Network 18: Reset Step No
   RUNG wire#powerrail
      Contact( "AlwaysTRUE" )
      wire#w1
      { S7_Templates := "SrcType := Int" } EQ_Contact(in1 := #STEP_NO, in2 := 11)
      I_Contact( #Modbus_Master_DB.MASTER_READ_DATA.MOD_COIL_DATA[14] )
      Contact( #ALL_FILL_DONE )
      wire#w2
      { S7_Templates := "time_type := Time" } #Step_Timer[12].TON(pt := t#0.5s, et =>)
      Move(in := 0, out1 => #STEP_NO)
   END_RUNG
   RUNG wire#w1
      { S7_Templates := "SrcType := Int" } EQ_Contact(in1 := #STEP_NO, in2 := 20)
      Contact( #ALL_FILL_DONE )
   END_RUNG wire#w2
   RUNG wire#w1
      Contact( #INxReset_Sequence )
   END_RUNG wire#w2
   RUNG wire#w1
      Contact( #INxReset_Sequence )
      R_Coil( #Filling_Done )
      R_Coil( #Cycle_Started )
      { S7_Templates := "SrcType := Real" } NE_Contact(in1 := #Gross_Weight, in2 := 0.0)
      wire#w3
      Move(in := 0.0, out1 => #Gross_Weight, out2 => #Net_Wieght, out3 => #Tare_Weight)
   END_RUNG
   RUNG wire#w3
      R_Coil( #Modbus_Master_DB.MASTER_WRITE_DATA.MOD_COIL_DATA[14] )
   END_RUNG
   // the same network as SCL:
   #Step_Timer[12].TON(IN := "AlwaysTRUE" AND (((#STEP_NO = 11) AND NOT #Modbus_Master_DB.MASTER_READ_DATA.MOD_COIL_DATA[14] AND #ALL_FILL_DONE) OR ((#STEP_NO = 20) AND #ALL_FILL_DONE) OR #INxReset_Sequence),
                       PT := t#0.5s);
   IF #Step_Timer[12].Q THEN #STEP_NO := 0; END_IF;
   #_w1 := "AlwaysTRUE" AND #INxReset_Sequence;
   IF #_w1 THEN
       #Filling_Done := FALSE;
       #Cycle_Started := FALSE;
   END_IF;
   #_w2 := #_w1 AND (#Gross_Weight <> 0.0);
   IF #_w2 THEN
       #Gross_Weight := 0.0;
       #Net_Wieght := 0.0;
       #Tare_Weight := 0.0;
       #Modbus_Master_DB.MASTER_WRITE_DATA.MOD_COIL_DATA[14] := FALSE;
   END_IF;
END_REGION

REGION Network 19: Output Mapping
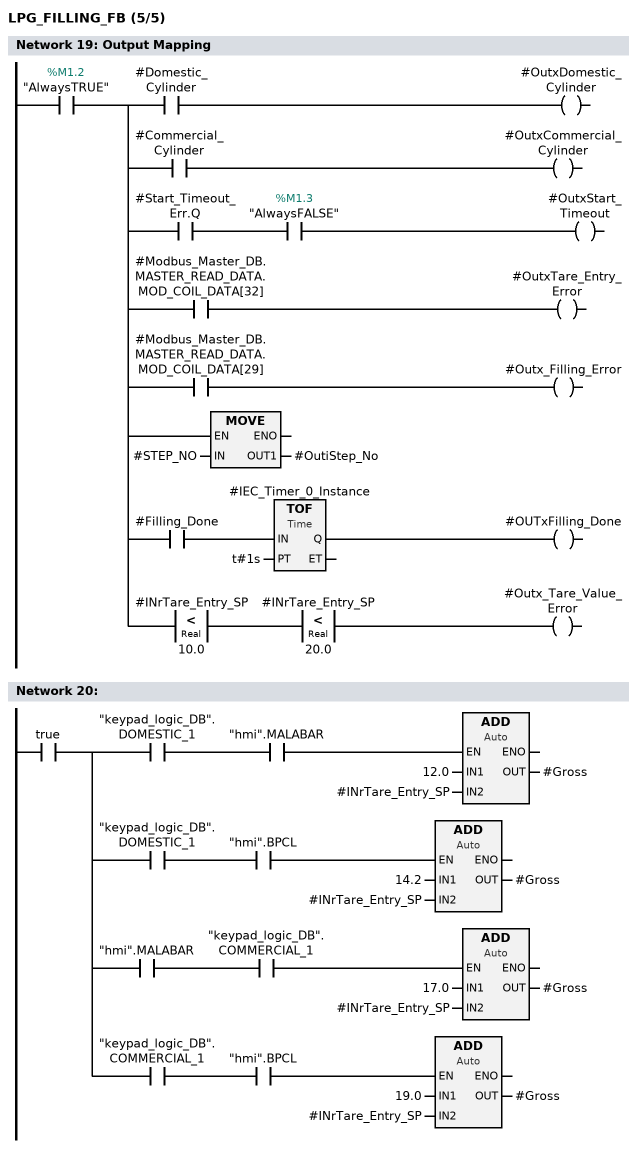
   RUNG wire#powerrail
      Contact( "AlwaysTRUE" )
      wire#w1
      Contact( #Domestic_Cylinder )
      Coil( #OutxDomestic_Cylinder )
   END_RUNG
   RUNG wire#w1
      Contact( #Commercial_Cylinder )
      Coil( #OutxCommercial_Cylinder )
   END_RUNG
   RUNG wire#w1
      Contact( #Start_Timeout_Err.Q )
      Contact( "AlwaysFALSE" )
      Coil( #OutxStart_Timeout )
   END_RUNG
   RUNG wire#w1
      Contact( #Modbus_Master_DB.MASTER_READ_DATA.MOD_COIL_DATA[32] )
      Coil( #OutxTare_Entry_Error )
   END_RUNG
   RUNG wire#w1
      Contact( #Modbus_Master_DB.MASTER_READ_DATA.MOD_COIL_DATA[29] )
      Coil( #Outx_Filling_Error )
   END_RUNG
   RUNG wire#w1
      Move(in := #STEP_NO, out1 => #OutiStep_No)
   END_RUNG
   RUNG wire#w1
      Contact( #Filling_Done )
      { S7_Templates := "time_type := Time" } #IEC_Timer_0_Instance.TOF(pt := t#1s, et =>)
      Coil( #OUTxFilling_Done )
   END_RUNG
   RUNG wire#w1
      { S7_Templates := "SrcType := Real" } LT_Contact(in1 := #INrTare_Entry_SP, in2 := 10.0)
      { S7_Templates := "SrcType := Real" } LT_Contact(in1 := #INrTare_Entry_SP, in2 := 20.0)
      Coil( #Outx_Tare_Value_Error )
   END_RUNG
   // the same network as SCL:
   #OutxDomestic_Cylinder := "AlwaysTRUE" AND #Domestic_Cylinder;
   #OutxCommercial_Cylinder := "AlwaysTRUE" AND #Commercial_Cylinder;
   #OutxStart_Timeout := "AlwaysTRUE" AND #Start_Timeout_Err.Q AND "AlwaysFALSE";
   #OutxTare_Entry_Error := "AlwaysTRUE" AND #Modbus_Master_DB.MASTER_READ_DATA.MOD_COIL_DATA[32];
   #Outx_Filling_Error := "AlwaysTRUE" AND #Modbus_Master_DB.MASTER_READ_DATA.MOD_COIL_DATA[29];
   IF "AlwaysTRUE" THEN #OutiStep_No := #STEP_NO; END_IF;
   #IEC_Timer_0_Instance(IN := "AlwaysTRUE" AND #Filling_Done, PT := t#1s);   // TOF
   #OUTxFilling_Done := #IEC_Timer_0_Instance.Q;
   #Outx_Tare_Value_Error := "AlwaysTRUE" AND (#INrTare_Entry_SP < 10.0) AND (#INrTare_Entry_SP < 20.0);
END_REGION

REGION Network 20
   RUNG wire#powerrail
      Contact( true )
      wire#w1
      Contact( "keypad_logic_DB".DOMESTIC_1 )
      Contact( "hmi".MALABAR )
      Add(in1 := 12.0, in2 := #INrTare_Entry_SP, out => #Gross)
   END_RUNG
   RUNG wire#w1
      Contact( "keypad_logic_DB".DOMESTIC_1 )
      Contact( "hmi".BPCL )
      Add(in1 := 14.2, in2 := #INrTare_Entry_SP, out => #Gross)
   END_RUNG
   RUNG wire#w1
      Contact( "hmi".MALABAR )
      Contact( "keypad_logic_DB".COMMERCIAL_1 )
      Add(in1 := 17.0, in2 := #INrTare_Entry_SP, out => #Gross)
   END_RUNG
   RUNG wire#w1
      Contact( "keypad_logic_DB".COMMERCIAL_1 )
      Contact( "hmi".BPCL )
      Add(in1 := 19.0, in2 := #INrTare_Entry_SP, out => #Gross)
   END_RUNG
   // the same network as SCL:
   IF true AND "keypad_logic_DB".DOMESTIC_1 AND "hmi".MALABAR THEN
       #Gross := 12.0 + #INrTare_Entry_SP;
   END_IF;
   IF true AND "keypad_logic_DB".DOMESTIC_1 AND "hmi".BPCL THEN #Gross := 14.2 + #INrTare_Entry_SP; END_IF;
   IF true AND "hmi".MALABAR AND "keypad_logic_DB".COMMERCIAL_1 THEN
       #Gross := 17.0 + #INrTare_Entry_SP;
   END_IF;
   IF true AND "keypad_logic_DB".COMMERCIAL_1 AND "hmi".BPCL THEN #Gross := 19.0 + #INrTare_Entry_SP; END_IF;
END_REGION
END_FUNCTION_BLOCK

FUNCTION_BLOCK "FILLING_STATION5_FB"   // FB501, LAD
{ S7_Optimized_Access := 'TRUE' }
VERSION : 0.1
// stored: AutoNumber false, IsIECCheckEnabled false, IsRetainMemResEnabled false, MemoryReserve 100, SetENOAutomatically false, UDAEnableTagReadback false
   VAR
      STATION5_S1 { S7_SetPoint := 'True'} : "LPG_FILLING_FB";
      STATION5_S2 { S7_SetPoint := 'True'} : "LPG_FILLING_FB";
      STATION5_S3 { S7_SetPoint := 'True'} : "LPG_FILLING_FB";
      STATION5_S4 { S7_SetPoint := 'True'} : "LPG_FILLING_FB";
      STATION5_S5 { S7_SetPoint := 'True'} : "LPG_FILLING_FB";
      STATION5_S6 { S7_SetPoint := 'True'} : "LPG_FILLING_FB";
      FILLING_STATION5 { S7_SetPoint := 'True'} : "FILLING_FB_L2";
      FILL_SEQ_STARTED_L2 { S7_SetPoint := 'True'} : Array[1..6] of Bool;
      FILLING_DONE_L2 : Array[1..6] of Bool;
   END_VAR
   VAR_TEMP   // added for the SCL form of the ladder/FBD networks
      _w1 : Bool;
   END_VAR
BEGIN

REGION Network 2: Call Filling Station-5 L2
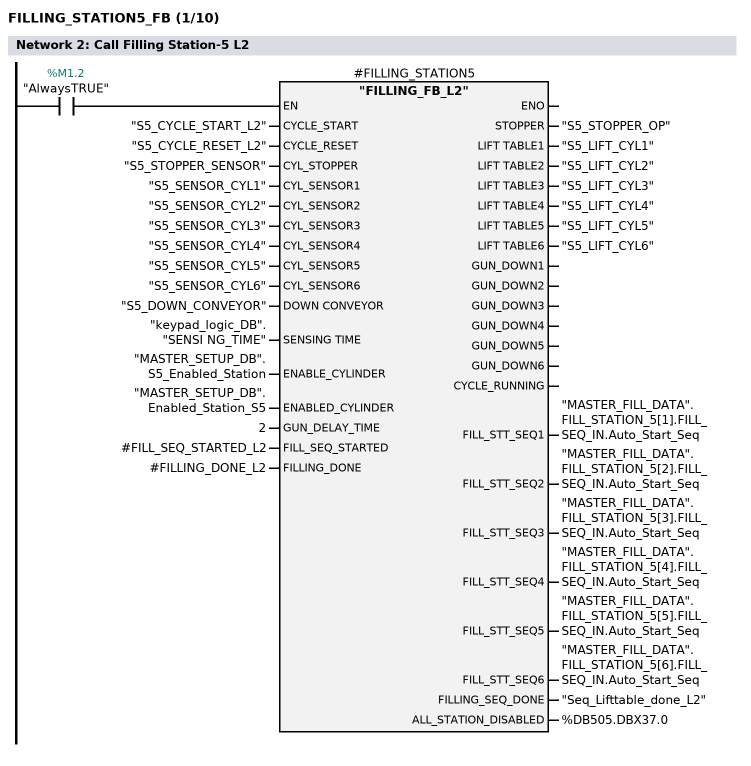
   RUNG wire#powerrail
      Contact( "AlwaysTRUE" )
      #FILLING_STATION5(CYCLE_START := "S5_CYCLE_START_L2", CYCLE_RESET := "S5_CYCLE_RESET_L2", CYL_STOPPER := "S5_STOPPER_SENSOR", CYL_SENSOR1 := "S5_SENSOR_CYL1", CYL_SENSOR2 := "S5_SENSOR_CYL2", CYL_SENSOR3 := "S5_SENSOR_CYL3", CYL_SENSOR4 := "S5_SENSOR_CYL4", CYL_SENSOR5 := "S5_SENSOR_CYL5", CYL_SENSOR6 := "S5_SENSOR_CYL6", "DOWN CONVEYOR" := "S5_DOWN_CONVEYOR", "SENSING TIME" := "keypad_logic_DB"."SENSI NG_TIME", ENABLE_CYLINDER := "MASTER_SETUP_DB".S5_Enabled_Station, ENABLED_CYLINDER := "MASTER_SETUP_DB".Enabled_Station_S5, GUN_DELAY_TIME := 2, FILL_SEQ_STARTED := #FILL_SEQ_STARTED_L2, FILLING_DONE := #FILLING_DONE_L2, STOPPER => "S5_STOPPER_OP", "LIFT TABLE1" => "S5_LIFT_CYL1", "LIFT TABLE2" => "S5_LIFT_CYL2", "LIFT TABLE3" => "S5_LIFT_CYL3", "LIFT TABLE4" => "S5_LIFT_CYL4", "LIFT TABLE5" => "S5_LIFT_CYL5", "LIFT TABLE6" => "S5_LIFT_CYL6", GUN_DOWN1 =>, GUN_DOWN2 =>, GUN_DOWN3 =>, GUN_DOWN4 =>, GUN_DOWN5 =>, GUN_DOWN6 =>, CYCLE_RUNNING =>, FILL_STT_SEQ1 => "MASTER_FILL_DATA".FILL_STATION_5[1].FILL_SEQ_IN.Auto_Start_Seq, FILL_STT_SEQ2 => "MASTER_FILL_DATA".FILL_STATION_5[2].FILL_SEQ_IN.Auto_Start_Seq, FILL_STT_SEQ3 => "MASTER_FILL_DATA".FILL_STATION_5[3].FILL_SEQ_IN.Auto_Start_Seq, FILL_STT_SEQ4 => "MASTER_FILL_DATA".FILL_STATION_5[4].FILL_SEQ_IN.Auto_Start_Seq, FILL_STT_SEQ5 => "MASTER_FILL_DATA".FILL_STATION_5[5].FILL_SEQ_IN.Auto_Start_Seq, FILL_STT_SEQ6 => "MASTER_FILL_DATA".FILL_STATION_5[6].FILL_SEQ_IN.Auto_Start_Seq, FILLING_SEQ_DONE => "Seq_Lifttable_done_L2", ALL_STATION_DISABLED => %DB505.DBX37.0)
   END_RUNG
   // the same network as SCL:
   IF "AlwaysTRUE" THEN
       #FILLING_STATION5(CYCLE_START := "S5_CYCLE_START_L2",   // "FILLING_FB_L2"
                         CYCLE_RESET := "S5_CYCLE_RESET_L2",
                         CYL_STOPPER := "S5_STOPPER_SENSOR",
                         CYL_SENSOR1 := "S5_SENSOR_CYL1",
                         CYL_SENSOR2 := "S5_SENSOR_CYL2",
                         CYL_SENSOR3 := "S5_SENSOR_CYL3",
                         CYL_SENSOR4 := "S5_SENSOR_CYL4",
                         CYL_SENSOR5 := "S5_SENSOR_CYL5",
                         CYL_SENSOR6 := "S5_SENSOR_CYL6",
                         "DOWN CONVEYOR" := "S5_DOWN_CONVEYOR",
                         "SENSING TIME" := "keypad_logic_DB"."SENSI NG_TIME",
                         ENABLE_CYLINDER := "MASTER_SETUP_DB".S5_Enabled_Station,
                         ENABLED_CYLINDER := "MASTER_SETUP_DB".Enabled_Station_S5,
                         GUN_DELAY_TIME := 2,
                         FILL_SEQ_STARTED := #FILL_SEQ_STARTED_L2,
                         FILLING_DONE := #FILLING_DONE_L2,
                         STOPPER => "S5_STOPPER_OP",
                         "LIFT TABLE1" => "S5_LIFT_CYL1",
                         "LIFT TABLE2" => "S5_LIFT_CYL2",
                         "LIFT TABLE3" => "S5_LIFT_CYL3",
                         "LIFT TABLE4" => "S5_LIFT_CYL4",
                         "LIFT TABLE5" => "S5_LIFT_CYL5",
                         "LIFT TABLE6" => "S5_LIFT_CYL6",
                         FILL_STT_SEQ1 => "MASTER_FILL_DATA".FILL_STATION_5[1].FILL_SEQ_IN.Auto_Start_Seq,
                         FILL_STT_SEQ2 => "MASTER_FILL_DATA".FILL_STATION_5[2].FILL_SEQ_IN.Auto_Start_Seq,
                         FILL_STT_SEQ3 => "MASTER_FILL_DATA".FILL_STATION_5[3].FILL_SEQ_IN.Auto_Start_Seq,
                         FILL_STT_SEQ4 => "MASTER_FILL_DATA".FILL_STATION_5[4].FILL_SEQ_IN.Auto_Start_Seq,
                         FILL_STT_SEQ5 => "MASTER_FILL_DATA".FILL_STATION_5[5].FILL_SEQ_IN.Auto_Start_Seq,
                         FILL_STT_SEQ6 => "MASTER_FILL_DATA".FILL_STATION_5[6].FILL_SEQ_IN.Auto_Start_Seq,
                         FILLING_SEQ_DONE => "Seq_Lifttable_done_L2",
                         ALL_STATION_DISABLED => %DB505.DBX37.0);
   END_IF;
END_REGION

REGION Network 3: Call Filling Line-1 Station-1 FB
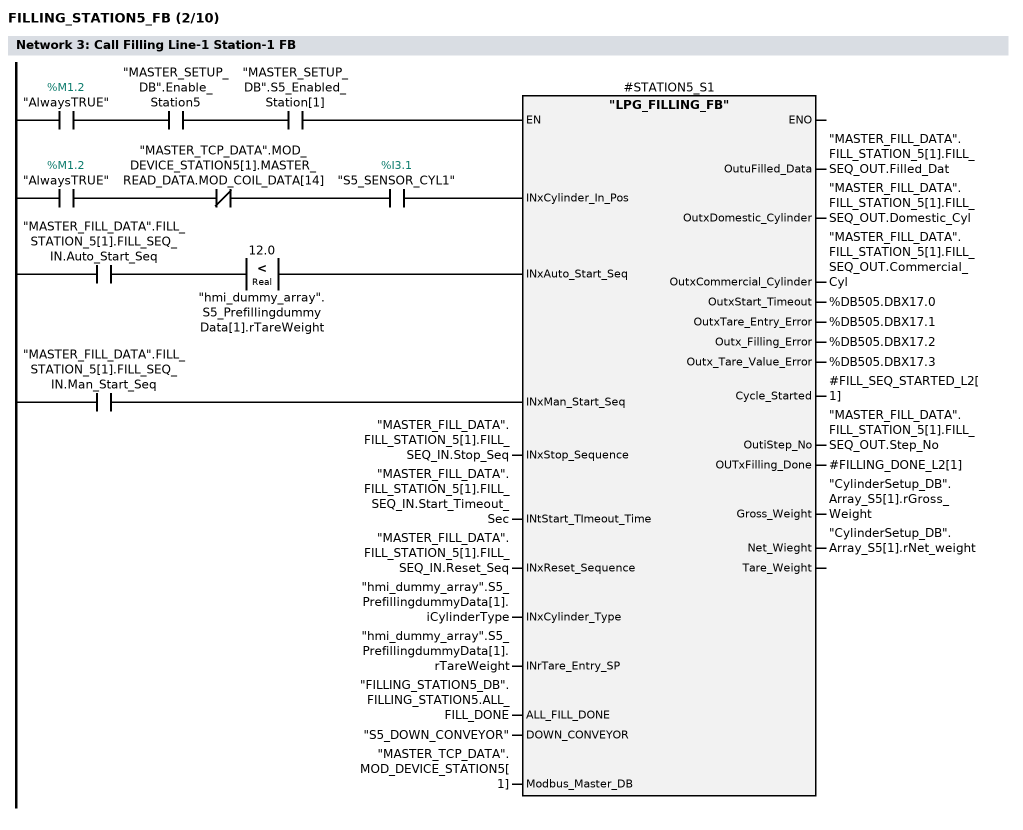
   RUNG wire#powerrail
      Contact( "AlwaysTRUE" )
      Contact( "MASTER_SETUP_DB".Enable_Station5 )
      Contact( "MASTER_SETUP_DB".S5_Enabled_Station[1] )
      #STATION5_S1(INxCylinder_In_Pos := wire#w1, INxAuto_Start_Seq := wire#w2, INxMan_Start_Seq := wire#w3, INxStop_Sequence := "MASTER_FILL_DATA".FILL_STATION_5[1].FILL_SEQ_IN.Stop_Seq, INtStart_TImeout_Time := "MASTER_FILL_DATA".FILL_STATION_5[1].FILL_SEQ_IN.Start_Timeout_Sec, INxReset_Sequence := "MASTER_FILL_DATA".FILL_STATION_5[1].FILL_SEQ_IN.Reset_Seq, INxCylinder_Type := "hmi_dummy_array".S5_PrefillingdummyData[1].iCylinderType, INrTare_Entry_SP := "hmi_dummy_array".S5_PrefillingdummyData[1].rTareWeight, ALL_FILL_DONE := "FILLING_STATION5_DB".FILLING_STATION5.ALL_FILL_DONE, DOWN_CONVEYOR := "S5_DOWN_CONVEYOR", Modbus_Master_DB := "MASTER_TCP_DATA".MOD_DEVICE_STATION5[1], OutuFilled_Data => "MASTER_FILL_DATA".FILL_STATION_5[1].FILL_SEQ_OUT.Filled_Dat, OutxDomestic_Cylinder => "MASTER_FILL_DATA".FILL_STATION_5[1].FILL_SEQ_OUT.Domestic_Cyl, OutxCommercial_Cylinder => "MASTER_FILL_DATA".FILL_STATION_5[1].FILL_SEQ_OUT.Commercial_Cyl, OutxStart_Timeout => %DB505.DBX17.0, OutxTare_Entry_Error => %DB505.DBX17.1, Outx_Filling_Error => %DB505.DBX17.2, Outx_Tare_Value_Error => %DB505.DBX17.3, Cycle_Started => #FILL_SEQ_STARTED_L2[1], OutiStep_No => "MASTER_FILL_DATA".FILL_STATION_5[1].FILL_SEQ_OUT.Step_No, OUTxFilling_Done => #FILLING_DONE_L2[1], Gross_Weight => "CylinderSetup_DB".Array_S5[1].rGross_Weight, Net_Wieght => "CylinderSetup_DB".Array_S5[1].rNet_weight, Tare_Weight =>)
   END_RUNG
   RUNG wire#powerrail
      Contact( "AlwaysTRUE" )
      I_Contact( "MASTER_TCP_DATA".MOD_DEVICE_STATION5[1].MASTER_READ_DATA.MOD_COIL_DATA[14] )
      Contact( "S5_SENSOR_CYL1" )
   END_RUNG wire#w1
   RUNG wire#powerrail
      Contact( "MASTER_FILL_DATA".FILL_STATION_5[1].FILL_SEQ_IN.Auto_Start_Seq )
      { S7_Templates := "SrcType := Real" } LT_Contact(in1 := 12.0, in2 := "hmi_dummy_array".S5_PrefillingdummyData[1].rTareWeight)
   END_RUNG wire#w2
   RUNG wire#powerrail
      Contact( "MASTER_FILL_DATA".FILL_STATION_5[1].FILL_SEQ_IN.Man_Start_Seq )
   END_RUNG wire#w3
   // the same network as SCL:
   IF "AlwaysTRUE" AND "MASTER_SETUP_DB".Enable_Station5 AND "MASTER_SETUP_DB".S5_Enabled_Station[1] THEN
       #STATION5_S1(INxCylinder_In_Pos := "AlwaysTRUE" AND NOT "MASTER_TCP_DATA".MOD_DEVICE_STATION5[1].MASTER_READ_DATA.MOD_COIL_DATA[14] AND "S5_SENSOR_CYL1",   // "LPG_FILLING_FB"
                    INxAuto_Start_Seq := "MASTER_FILL_DATA".FILL_STATION_5[1].FILL_SEQ_IN.Auto_Start_Seq AND (12.0 < "hmi_dummy_array".S5_PrefillingdummyData[1].rTareWeight),
                    INxMan_Start_Seq := "MASTER_FILL_DATA".FILL_STATION_5[1].FILL_SEQ_IN.Man_Start_Seq,
                    INxStop_Sequence := "MASTER_FILL_DATA".FILL_STATION_5[1].FILL_SEQ_IN.Stop_Seq,
                    INtStart_TImeout_Time := "MASTER_FILL_DATA".FILL_STATION_5[1].FILL_SEQ_IN.Start_Timeout_Sec,
                    INxReset_Sequence := "MASTER_FILL_DATA".FILL_STATION_5[1].FILL_SEQ_IN.Reset_Seq,
                    INxCylinder_Type := "hmi_dummy_array".S5_PrefillingdummyData[1].iCylinderType,
                    INrTare_Entry_SP := "hmi_dummy_array".S5_PrefillingdummyData[1].rTareWeight,
                    ALL_FILL_DONE := "FILLING_STATION5_DB".FILLING_STATION5.ALL_FILL_DONE,
                    DOWN_CONVEYOR := "S5_DOWN_CONVEYOR",
                    Modbus_Master_DB := "MASTER_TCP_DATA".MOD_DEVICE_STATION5[1],
                    OutuFilled_Data => "MASTER_FILL_DATA".FILL_STATION_5[1].FILL_SEQ_OUT.Filled_Dat,
                    OutxDomestic_Cylinder => "MASTER_FILL_DATA".FILL_STATION_5[1].FILL_SEQ_OUT.Domestic_Cyl,
                    OutxCommercial_Cylinder => "MASTER_FILL_DATA".FILL_STATION_5[1].FILL_SEQ_OUT.Commercial_Cyl,
                    OutxStart_Timeout => %DB505.DBX17.0,
                    OutxTare_Entry_Error => %DB505.DBX17.1,
                    Outx_Filling_Error => %DB505.DBX17.2,
                    Outx_Tare_Value_Error => %DB505.DBX17.3,
                    Cycle_Started => #FILL_SEQ_STARTED_L2[1],
                    OutiStep_No => "MASTER_FILL_DATA".FILL_STATION_5[1].FILL_SEQ_OUT.Step_No,
                    OUTxFilling_Done => #FILLING_DONE_L2[1],
                    Gross_Weight => "CylinderSetup_DB".Array_S5[1].rGross_Weight,
                    Net_Wieght => "CylinderSetup_DB".Array_S5[1].rNet_weight);
   END_IF;
END_REGION

REGION Network 4: Call Filling Line-1 Station-2 FB
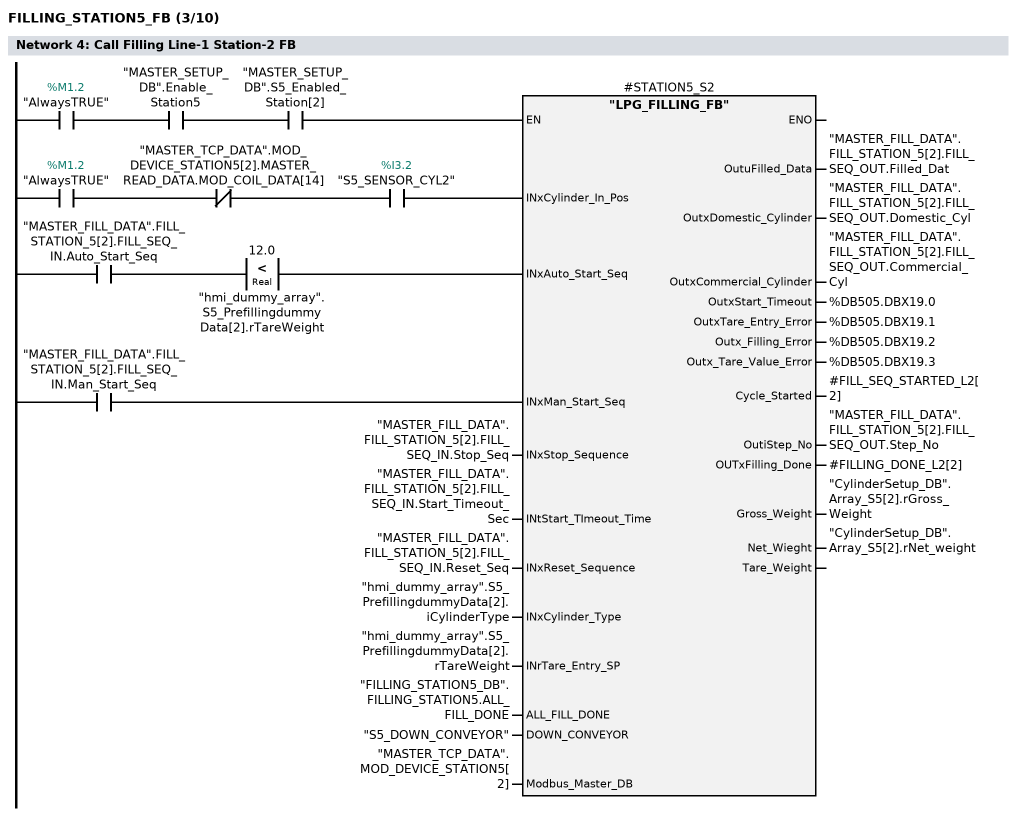
   RUNG wire#powerrail
      Contact( "AlwaysTRUE" )
      Contact( "MASTER_SETUP_DB".Enable_Station5 )
      Contact( "MASTER_SETUP_DB".S5_Enabled_Station[2] )
      #STATION5_S2(INxCylinder_In_Pos := wire#w1, INxAuto_Start_Seq := wire#w2, INxMan_Start_Seq := wire#w3, INxStop_Sequence := "MASTER_FILL_DATA".FILL_STATION_5[2].FILL_SEQ_IN.Stop_Seq, INtStart_TImeout_Time := "MASTER_FILL_DATA".FILL_STATION_5[2].FILL_SEQ_IN.Start_Timeout_Sec, INxReset_Sequence := "MASTER_FILL_DATA".FILL_STATION_5[2].FILL_SEQ_IN.Reset_Seq, INxCylinder_Type := "hmi_dummy_array".S5_PrefillingdummyData[2].iCylinderType, INrTare_Entry_SP := "hmi_dummy_array".S5_PrefillingdummyData[2].rTareWeight, ALL_FILL_DONE := "FILLING_STATION5_DB".FILLING_STATION5.ALL_FILL_DONE, DOWN_CONVEYOR := "S5_DOWN_CONVEYOR", Modbus_Master_DB := "MASTER_TCP_DATA".MOD_DEVICE_STATION5[2], OutuFilled_Data => "MASTER_FILL_DATA".FILL_STATION_5[2].FILL_SEQ_OUT.Filled_Dat, OutxDomestic_Cylinder => "MASTER_FILL_DATA".FILL_STATION_5[2].FILL_SEQ_OUT.Domestic_Cyl, OutxCommercial_Cylinder => "MASTER_FILL_DATA".FILL_STATION_5[2].FILL_SEQ_OUT.Commercial_Cyl, OutxStart_Timeout => %DB505.DBX19.0, OutxTare_Entry_Error => %DB505.DBX19.1, Outx_Filling_Error => %DB505.DBX19.2, Outx_Tare_Value_Error => %DB505.DBX19.3, Cycle_Started => #FILL_SEQ_STARTED_L2[2], OutiStep_No => "MASTER_FILL_DATA".FILL_STATION_5[2].FILL_SEQ_OUT.Step_No, OUTxFilling_Done => #FILLING_DONE_L2[2], Gross_Weight => "CylinderSetup_DB".Array_S5[2].rGross_Weight, Net_Wieght => "CylinderSetup_DB".Array_S5[2].rNet_weight, Tare_Weight =>)
   END_RUNG
   RUNG wire#powerrail
      Contact( "AlwaysTRUE" )
      I_Contact( "MASTER_TCP_DATA".MOD_DEVICE_STATION5[2].MASTER_READ_DATA.MOD_COIL_DATA[14] )
      Contact( "S5_SENSOR_CYL2" )
   END_RUNG wire#w1
   RUNG wire#powerrail
      Contact( "MASTER_FILL_DATA".FILL_STATION_5[2].FILL_SEQ_IN.Auto_Start_Seq )
      { S7_Templates := "SrcType := Real" } LT_Contact(in1 := 12.0, in2 := "hmi_dummy_array".S5_PrefillingdummyData[2].rTareWeight)
   END_RUNG wire#w2
   RUNG wire#powerrail
      Contact( "MASTER_FILL_DATA".FILL_STATION_5[2].FILL_SEQ_IN.Man_Start_Seq )
   END_RUNG wire#w3
   // the same network as SCL:
   IF "AlwaysTRUE" AND "MASTER_SETUP_DB".Enable_Station5 AND "MASTER_SETUP_DB".S5_Enabled_Station[2] THEN
       #STATION5_S2(INxCylinder_In_Pos := "AlwaysTRUE" AND NOT "MASTER_TCP_DATA".MOD_DEVICE_STATION5[2].MASTER_READ_DATA.MOD_COIL_DATA[14] AND "S5_SENSOR_CYL2",   // "LPG_FILLING_FB"
                    INxAuto_Start_Seq := "MASTER_FILL_DATA".FILL_STATION_5[2].FILL_SEQ_IN.Auto_Start_Seq AND (12.0 < "hmi_dummy_array".S5_PrefillingdummyData[2].rTareWeight),
                    INxMan_Start_Seq := "MASTER_FILL_DATA".FILL_STATION_5[2].FILL_SEQ_IN.Man_Start_Seq,
                    INxStop_Sequence := "MASTER_FILL_DATA".FILL_STATION_5[2].FILL_SEQ_IN.Stop_Seq,
                    INtStart_TImeout_Time := "MASTER_FILL_DATA".FILL_STATION_5[2].FILL_SEQ_IN.Start_Timeout_Sec,
                    INxReset_Sequence := "MASTER_FILL_DATA".FILL_STATION_5[2].FILL_SEQ_IN.Reset_Seq,
                    INxCylinder_Type := "hmi_dummy_array".S5_PrefillingdummyData[2].iCylinderType,
                    INrTare_Entry_SP := "hmi_dummy_array".S5_PrefillingdummyData[2].rTareWeight,
                    ALL_FILL_DONE := "FILLING_STATION5_DB".FILLING_STATION5.ALL_FILL_DONE,
                    DOWN_CONVEYOR := "S5_DOWN_CONVEYOR",
                    Modbus_Master_DB := "MASTER_TCP_DATA".MOD_DEVICE_STATION5[2],
                    OutuFilled_Data => "MASTER_FILL_DATA".FILL_STATION_5[2].FILL_SEQ_OUT.Filled_Dat,
                    OutxDomestic_Cylinder => "MASTER_FILL_DATA".FILL_STATION_5[2].FILL_SEQ_OUT.Domestic_Cyl,
                    OutxCommercial_Cylinder => "MASTER_FILL_DATA".FILL_STATION_5[2].FILL_SEQ_OUT.Commercial_Cyl,
                    OutxStart_Timeout => %DB505.DBX19.0,
                    OutxTare_Entry_Error => %DB505.DBX19.1,
                    Outx_Filling_Error => %DB505.DBX19.2,
                    Outx_Tare_Value_Error => %DB505.DBX19.3,
                    Cycle_Started => #FILL_SEQ_STARTED_L2[2],
                    OutiStep_No => "MASTER_FILL_DATA".FILL_STATION_5[2].FILL_SEQ_OUT.Step_No,
                    OUTxFilling_Done => #FILLING_DONE_L2[2],
                    Gross_Weight => "CylinderSetup_DB".Array_S5[2].rGross_Weight,
                    Net_Wieght => "CylinderSetup_DB".Array_S5[2].rNet_weight);
   END_IF;
END_REGION

REGION Network 5: Call Filling Line-1 Station-3 FB
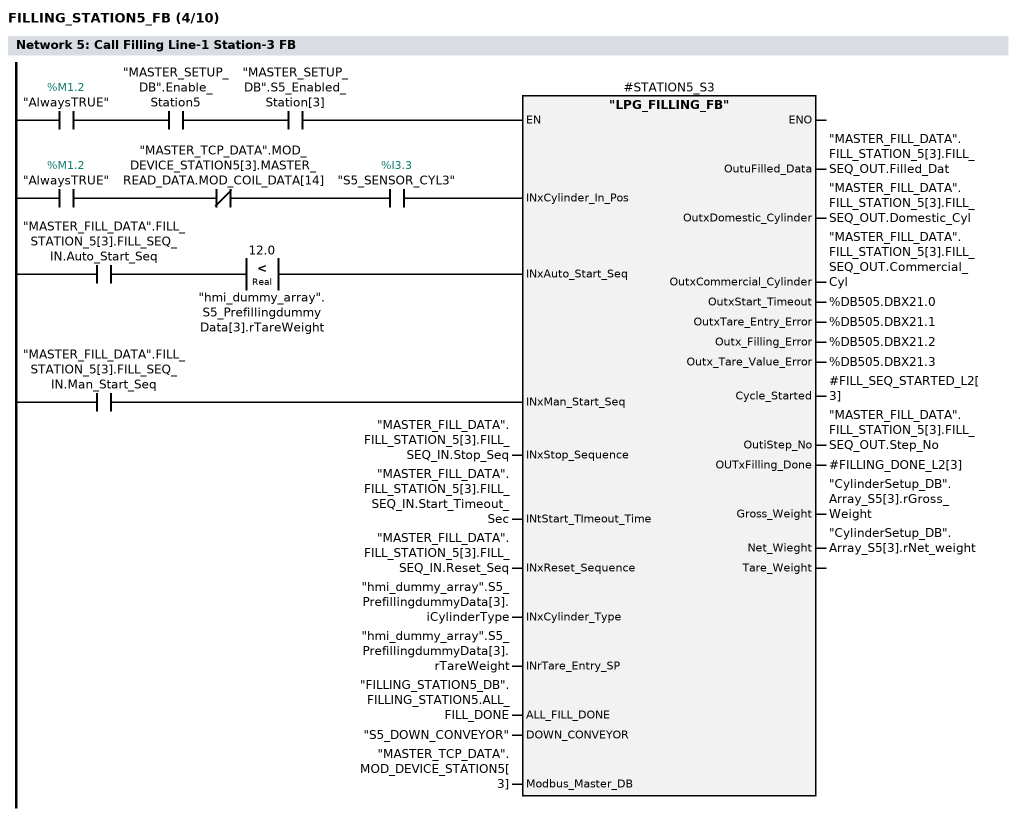
   RUNG wire#powerrail
      Contact( "AlwaysTRUE" )
      Contact( "MASTER_SETUP_DB".Enable_Station5 )
      Contact( "MASTER_SETUP_DB".S5_Enabled_Station[3] )
      #STATION5_S3(INxCylinder_In_Pos := wire#w1, INxAuto_Start_Seq := wire#w2, INxMan_Start_Seq := wire#w3, INxStop_Sequence := "MASTER_FILL_DATA".FILL_STATION_5[3].FILL_SEQ_IN.Stop_Seq, INtStart_TImeout_Time := "MASTER_FILL_DATA".FILL_STATION_5[3].FILL_SEQ_IN.Start_Timeout_Sec, INxReset_Sequence := "MASTER_FILL_DATA".FILL_STATION_5[3].FILL_SEQ_IN.Reset_Seq, INxCylinder_Type := "hmi_dummy_array".S5_PrefillingdummyData[3].iCylinderType, INrTare_Entry_SP := "hmi_dummy_array".S5_PrefillingdummyData[3].rTareWeight, ALL_FILL_DONE := "FILLING_STATION5_DB".FILLING_STATION5.ALL_FILL_DONE, DOWN_CONVEYOR := "S5_DOWN_CONVEYOR", Modbus_Master_DB := "MASTER_TCP_DATA".MOD_DEVICE_STATION5[3], OutuFilled_Data => "MASTER_FILL_DATA".FILL_STATION_5[3].FILL_SEQ_OUT.Filled_Dat, OutxDomestic_Cylinder => "MASTER_FILL_DATA".FILL_STATION_5[3].FILL_SEQ_OUT.Domestic_Cyl, OutxCommercial_Cylinder => "MASTER_FILL_DATA".FILL_STATION_5[3].FILL_SEQ_OUT.Commercial_Cyl, OutxStart_Timeout => %DB505.DBX21.0, OutxTare_Entry_Error => %DB505.DBX21.1, Outx_Filling_Error => %DB505.DBX21.2, Outx_Tare_Value_Error => %DB505.DBX21.3, Cycle_Started => #FILL_SEQ_STARTED_L2[3], OutiStep_No => "MASTER_FILL_DATA".FILL_STATION_5[3].FILL_SEQ_OUT.Step_No, OUTxFilling_Done => #FILLING_DONE_L2[3], Gross_Weight => "CylinderSetup_DB".Array_S5[3].rGross_Weight, Net_Wieght => "CylinderSetup_DB".Array_S5[3].rNet_weight, Tare_Weight =>)
   END_RUNG
   RUNG wire#powerrail
      Contact( "AlwaysTRUE" )
      I_Contact( "MASTER_TCP_DATA".MOD_DEVICE_STATION5[3].MASTER_READ_DATA.MOD_COIL_DATA[14] )
      Contact( "S5_SENSOR_CYL3" )
   END_RUNG wire#w1
   RUNG wire#powerrail
      Contact( "MASTER_FILL_DATA".FILL_STATION_5[3].FILL_SEQ_IN.Auto_Start_Seq )
      { S7_Templates := "SrcType := Real" } LT_Contact(in1 := 12.0, in2 := "hmi_dummy_array".S5_PrefillingdummyData[3].rTareWeight)
   END_RUNG wire#w2
   RUNG wire#powerrail
      Contact( "MASTER_FILL_DATA".FILL_STATION_5[3].FILL_SEQ_IN.Man_Start_Seq )
   END_RUNG wire#w3
   // the same network as SCL:
   IF "AlwaysTRUE" AND "MASTER_SETUP_DB".Enable_Station5 AND "MASTER_SETUP_DB".S5_Enabled_Station[3] THEN
       #STATION5_S3(INxCylinder_In_Pos := "AlwaysTRUE" AND NOT "MASTER_TCP_DATA".MOD_DEVICE_STATION5[3].MASTER_READ_DATA.MOD_COIL_DATA[14] AND "S5_SENSOR_CYL3",   // "LPG_FILLING_FB"
                    INxAuto_Start_Seq := "MASTER_FILL_DATA".FILL_STATION_5[3].FILL_SEQ_IN.Auto_Start_Seq AND (12.0 < "hmi_dummy_array".S5_PrefillingdummyData[3].rTareWeight),
                    INxMan_Start_Seq := "MASTER_FILL_DATA".FILL_STATION_5[3].FILL_SEQ_IN.Man_Start_Seq,
                    INxStop_Sequence := "MASTER_FILL_DATA".FILL_STATION_5[3].FILL_SEQ_IN.Stop_Seq,
                    INtStart_TImeout_Time := "MASTER_FILL_DATA".FILL_STATION_5[3].FILL_SEQ_IN.Start_Timeout_Sec,
                    INxReset_Sequence := "MASTER_FILL_DATA".FILL_STATION_5[3].FILL_SEQ_IN.Reset_Seq,
                    INxCylinder_Type := "hmi_dummy_array".S5_PrefillingdummyData[3].iCylinderType,
                    INrTare_Entry_SP := "hmi_dummy_array".S5_PrefillingdummyData[3].rTareWeight,
                    ALL_FILL_DONE := "FILLING_STATION5_DB".FILLING_STATION5.ALL_FILL_DONE,
                    DOWN_CONVEYOR := "S5_DOWN_CONVEYOR",
                    Modbus_Master_DB := "MASTER_TCP_DATA".MOD_DEVICE_STATION5[3],
                    OutuFilled_Data => "MASTER_FILL_DATA".FILL_STATION_5[3].FILL_SEQ_OUT.Filled_Dat,
                    OutxDomestic_Cylinder => "MASTER_FILL_DATA".FILL_STATION_5[3].FILL_SEQ_OUT.Domestic_Cyl,
                    OutxCommercial_Cylinder => "MASTER_FILL_DATA".FILL_STATION_5[3].FILL_SEQ_OUT.Commercial_Cyl,
                    OutxStart_Timeout => %DB505.DBX21.0,
                    OutxTare_Entry_Error => %DB505.DBX21.1,
                    Outx_Filling_Error => %DB505.DBX21.2,
                    Outx_Tare_Value_Error => %DB505.DBX21.3,
                    Cycle_Started => #FILL_SEQ_STARTED_L2[3],
                    OutiStep_No => "MASTER_FILL_DATA".FILL_STATION_5[3].FILL_SEQ_OUT.Step_No,
                    OUTxFilling_Done => #FILLING_DONE_L2[3],
                    Gross_Weight => "CylinderSetup_DB".Array_S5[3].rGross_Weight,
                    Net_Wieght => "CylinderSetup_DB".Array_S5[3].rNet_weight);
   END_IF;
END_REGION

REGION Network 6: Call Filling Line-1 Station-4 FB
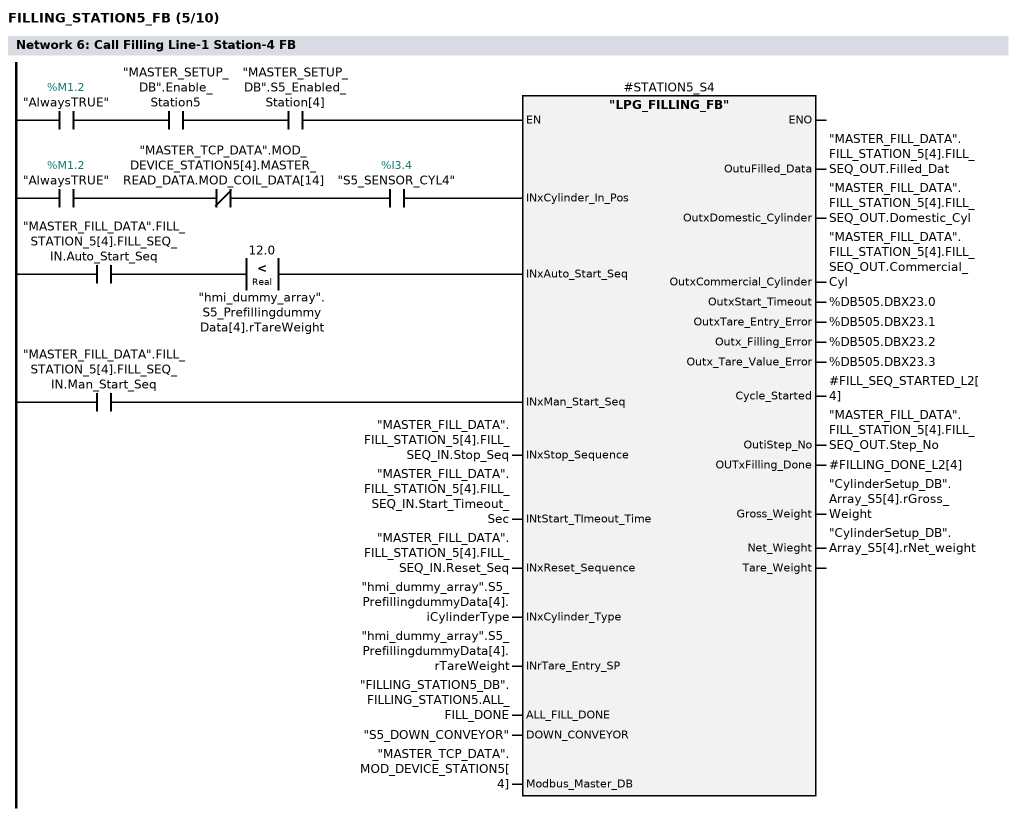
   RUNG wire#powerrail
      Contact( "AlwaysTRUE" )
      Contact( "MASTER_SETUP_DB".Enable_Station5 )
      Contact( "MASTER_SETUP_DB".S5_Enabled_Station[4] )
      #STATION5_S4(INxCylinder_In_Pos := wire#w1, INxAuto_Start_Seq := wire#w2, INxMan_Start_Seq := wire#w3, INxStop_Sequence := "MASTER_FILL_DATA".FILL_STATION_5[4].FILL_SEQ_IN.Stop_Seq, INtStart_TImeout_Time := "MASTER_FILL_DATA".FILL_STATION_5[4].FILL_SEQ_IN.Start_Timeout_Sec, INxReset_Sequence := "MASTER_FILL_DATA".FILL_STATION_5[4].FILL_SEQ_IN.Reset_Seq, INxCylinder_Type := "hmi_dummy_array".S5_PrefillingdummyData[4].iCylinderType, INrTare_Entry_SP := "hmi_dummy_array".S5_PrefillingdummyData[4].rTareWeight, ALL_FILL_DONE := "FILLING_STATION5_DB".FILLING_STATION5.ALL_FILL_DONE, DOWN_CONVEYOR := "S5_DOWN_CONVEYOR", Modbus_Master_DB := "MASTER_TCP_DATA".MOD_DEVICE_STATION5[4], OutuFilled_Data => "MASTER_FILL_DATA".FILL_STATION_5[4].FILL_SEQ_OUT.Filled_Dat, OutxDomestic_Cylinder => "MASTER_FILL_DATA".FILL_STATION_5[4].FILL_SEQ_OUT.Domestic_Cyl, OutxCommercial_Cylinder => "MASTER_FILL_DATA".FILL_STATION_5[4].FILL_SEQ_OUT.Commercial_Cyl, OutxStart_Timeout => %DB505.DBX23.0, OutxTare_Entry_Error => %DB505.DBX23.1, Outx_Filling_Error => %DB505.DBX23.2, Outx_Tare_Value_Error => %DB505.DBX23.3, Cycle_Started => #FILL_SEQ_STARTED_L2[4], OutiStep_No => "MASTER_FILL_DATA".FILL_STATION_5[4].FILL_SEQ_OUT.Step_No, OUTxFilling_Done => #FILLING_DONE_L2[4], Gross_Weight => "CylinderSetup_DB".Array_S5[4].rGross_Weight, Net_Wieght => "CylinderSetup_DB".Array_S5[4].rNet_weight, Tare_Weight =>)
   END_RUNG
   RUNG wire#powerrail
      Contact( "AlwaysTRUE" )
      I_Contact( "MASTER_TCP_DATA".MOD_DEVICE_STATION5[4].MASTER_READ_DATA.MOD_COIL_DATA[14] )
      Contact( "S5_SENSOR_CYL4" )
   END_RUNG wire#w1
   RUNG wire#powerrail
      Contact( "MASTER_FILL_DATA".FILL_STATION_5[4].FILL_SEQ_IN.Auto_Start_Seq )
      { S7_Templates := "SrcType := Real" } LT_Contact(in1 := 12.0, in2 := "hmi_dummy_array".S5_PrefillingdummyData[4].rTareWeight)
   END_RUNG wire#w2
   RUNG wire#powerrail
      Contact( "MASTER_FILL_DATA".FILL_STATION_5[4].FILL_SEQ_IN.Man_Start_Seq )
   END_RUNG wire#w3
   // the same network as SCL:
   IF "AlwaysTRUE" AND "MASTER_SETUP_DB".Enable_Station5 AND "MASTER_SETUP_DB".S5_Enabled_Station[4] THEN
       #STATION5_S4(INxCylinder_In_Pos := "AlwaysTRUE" AND NOT "MASTER_TCP_DATA".MOD_DEVICE_STATION5[4].MASTER_READ_DATA.MOD_COIL_DATA[14] AND "S5_SENSOR_CYL4",   // "LPG_FILLING_FB"
                    INxAuto_Start_Seq := "MASTER_FILL_DATA".FILL_STATION_5[4].FILL_SEQ_IN.Auto_Start_Seq AND (12.0 < "hmi_dummy_array".S5_PrefillingdummyData[4].rTareWeight),
                    INxMan_Start_Seq := "MASTER_FILL_DATA".FILL_STATION_5[4].FILL_SEQ_IN.Man_Start_Seq,
                    INxStop_Sequence := "MASTER_FILL_DATA".FILL_STATION_5[4].FILL_SEQ_IN.Stop_Seq,
                    INtStart_TImeout_Time := "MASTER_FILL_DATA".FILL_STATION_5[4].FILL_SEQ_IN.Start_Timeout_Sec,
                    INxReset_Sequence := "MASTER_FILL_DATA".FILL_STATION_5[4].FILL_SEQ_IN.Reset_Seq,
                    INxCylinder_Type := "hmi_dummy_array".S5_PrefillingdummyData[4].iCylinderType,
                    INrTare_Entry_SP := "hmi_dummy_array".S5_PrefillingdummyData[4].rTareWeight,
                    ALL_FILL_DONE := "FILLING_STATION5_DB".FILLING_STATION5.ALL_FILL_DONE,
                    DOWN_CONVEYOR := "S5_DOWN_CONVEYOR",
                    Modbus_Master_DB := "MASTER_TCP_DATA".MOD_DEVICE_STATION5[4],
                    OutuFilled_Data => "MASTER_FILL_DATA".FILL_STATION_5[4].FILL_SEQ_OUT.Filled_Dat,
                    OutxDomestic_Cylinder => "MASTER_FILL_DATA".FILL_STATION_5[4].FILL_SEQ_OUT.Domestic_Cyl,
                    OutxCommercial_Cylinder => "MASTER_FILL_DATA".FILL_STATION_5[4].FILL_SEQ_OUT.Commercial_Cyl,
                    OutxStart_Timeout => %DB505.DBX23.0,
                    OutxTare_Entry_Error => %DB505.DBX23.1,
                    Outx_Filling_Error => %DB505.DBX23.2,
                    Outx_Tare_Value_Error => %DB505.DBX23.3,
                    Cycle_Started => #FILL_SEQ_STARTED_L2[4],
                    OutiStep_No => "MASTER_FILL_DATA".FILL_STATION_5[4].FILL_SEQ_OUT.Step_No,
                    OUTxFilling_Done => #FILLING_DONE_L2[4],
                    Gross_Weight => "CylinderSetup_DB".Array_S5[4].rGross_Weight,
                    Net_Wieght => "CylinderSetup_DB".Array_S5[4].rNet_weight);
   END_IF;
END_REGION

REGION Network 7: Call Filling Line-1 Station-5 FB
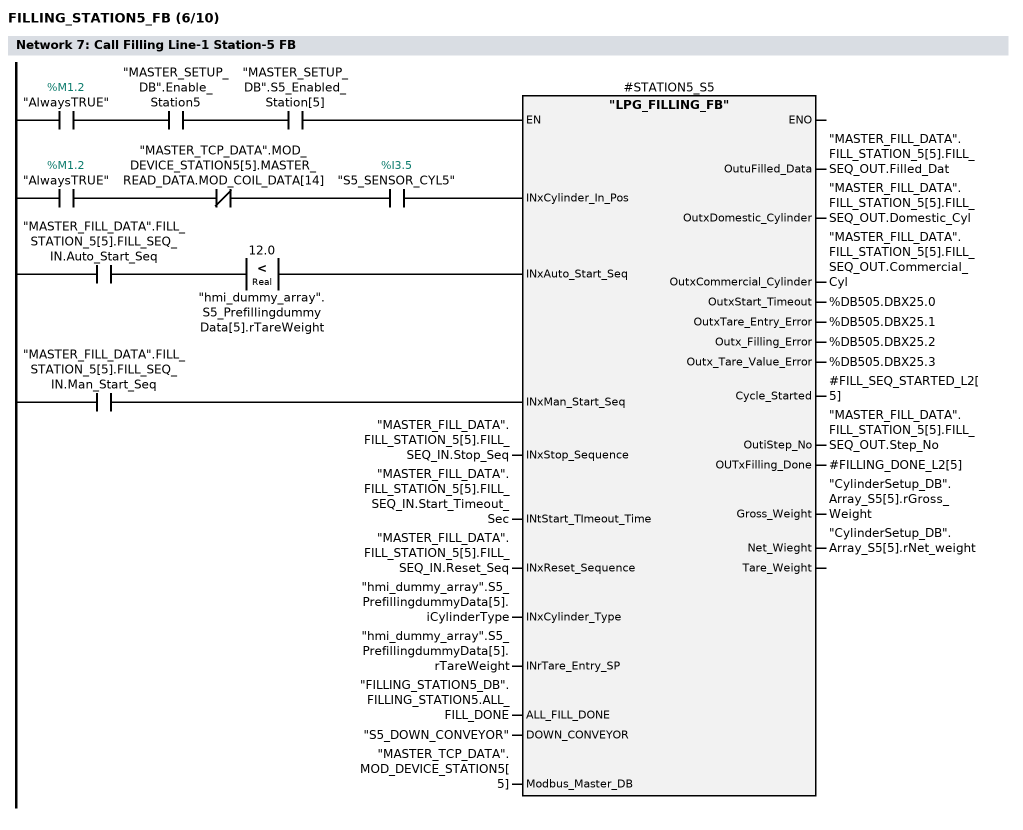
   RUNG wire#powerrail
      Contact( "AlwaysTRUE" )
      Contact( "MASTER_SETUP_DB".Enable_Station5 )
      Contact( "MASTER_SETUP_DB".S5_Enabled_Station[5] )
      #STATION5_S5(INxCylinder_In_Pos := wire#w1, INxAuto_Start_Seq := wire#w2, INxMan_Start_Seq := wire#w3, INxStop_Sequence := "MASTER_FILL_DATA".FILL_STATION_5[5].FILL_SEQ_IN.Stop_Seq, INtStart_TImeout_Time := "MASTER_FILL_DATA".FILL_STATION_5[5].FILL_SEQ_IN.Start_Timeout_Sec, INxReset_Sequence := "MASTER_FILL_DATA".FILL_STATION_5[5].FILL_SEQ_IN.Reset_Seq, INxCylinder_Type := "hmi_dummy_array".S5_PrefillingdummyData[5].iCylinderType, INrTare_Entry_SP := "hmi_dummy_array".S5_PrefillingdummyData[5].rTareWeight, ALL_FILL_DONE := "FILLING_STATION5_DB".FILLING_STATION5.ALL_FILL_DONE, DOWN_CONVEYOR := "S5_DOWN_CONVEYOR", Modbus_Master_DB := "MASTER_TCP_DATA".MOD_DEVICE_STATION5[5], OutuFilled_Data => "MASTER_FILL_DATA".FILL_STATION_5[5].FILL_SEQ_OUT.Filled_Dat, OutxDomestic_Cylinder => "MASTER_FILL_DATA".FILL_STATION_5[5].FILL_SEQ_OUT.Domestic_Cyl, OutxCommercial_Cylinder => "MASTER_FILL_DATA".FILL_STATION_5[5].FILL_SEQ_OUT.Commercial_Cyl, OutxStart_Timeout => %DB505.DBX25.0, OutxTare_Entry_Error => %DB505.DBX25.1, Outx_Filling_Error => %DB505.DBX25.2, Outx_Tare_Value_Error => %DB505.DBX25.3, Cycle_Started => #FILL_SEQ_STARTED_L2[5], OutiStep_No => "MASTER_FILL_DATA".FILL_STATION_5[5].FILL_SEQ_OUT.Step_No, OUTxFilling_Done => #FILLING_DONE_L2[5], Gross_Weight => "CylinderSetup_DB".Array_S5[5].rGross_Weight, Net_Wieght => "CylinderSetup_DB".Array_S5[5].rNet_weight, Tare_Weight =>)
   END_RUNG
   RUNG wire#powerrail
      Contact( "AlwaysTRUE" )
      I_Contact( "MASTER_TCP_DATA".MOD_DEVICE_STATION5[5].MASTER_READ_DATA.MOD_COIL_DATA[14] )
      Contact( "S5_SENSOR_CYL5" )
   END_RUNG wire#w1
   RUNG wire#powerrail
      Contact( "MASTER_FILL_DATA".FILL_STATION_5[5].FILL_SEQ_IN.Auto_Start_Seq )
      { S7_Templates := "SrcType := Real" } LT_Contact(in1 := 12.0, in2 := "hmi_dummy_array".S5_PrefillingdummyData[5].rTareWeight)
   END_RUNG wire#w2
   RUNG wire#powerrail
      Contact( "MASTER_FILL_DATA".FILL_STATION_5[5].FILL_SEQ_IN.Man_Start_Seq )
   END_RUNG wire#w3
   // the same network as SCL:
   IF "AlwaysTRUE" AND "MASTER_SETUP_DB".Enable_Station5 AND "MASTER_SETUP_DB".S5_Enabled_Station[5] THEN
       #STATION5_S5(INxCylinder_In_Pos := "AlwaysTRUE" AND NOT "MASTER_TCP_DATA".MOD_DEVICE_STATION5[5].MASTER_READ_DATA.MOD_COIL_DATA[14] AND "S5_SENSOR_CYL5",   // "LPG_FILLING_FB"
                    INxAuto_Start_Seq := "MASTER_FILL_DATA".FILL_STATION_5[5].FILL_SEQ_IN.Auto_Start_Seq AND (12.0 < "hmi_dummy_array".S5_PrefillingdummyData[5].rTareWeight),
                    INxMan_Start_Seq := "MASTER_FILL_DATA".FILL_STATION_5[5].FILL_SEQ_IN.Man_Start_Seq,
                    INxStop_Sequence := "MASTER_FILL_DATA".FILL_STATION_5[5].FILL_SEQ_IN.Stop_Seq,
                    INtStart_TImeout_Time := "MASTER_FILL_DATA".FILL_STATION_5[5].FILL_SEQ_IN.Start_Timeout_Sec,
                    INxReset_Sequence := "MASTER_FILL_DATA".FILL_STATION_5[5].FILL_SEQ_IN.Reset_Seq,
                    INxCylinder_Type := "hmi_dummy_array".S5_PrefillingdummyData[5].iCylinderType,
                    INrTare_Entry_SP := "hmi_dummy_array".S5_PrefillingdummyData[5].rTareWeight,
                    ALL_FILL_DONE := "FILLING_STATION5_DB".FILLING_STATION5.ALL_FILL_DONE,
                    DOWN_CONVEYOR := "S5_DOWN_CONVEYOR",
                    Modbus_Master_DB := "MASTER_TCP_DATA".MOD_DEVICE_STATION5[5],
                    OutuFilled_Data => "MASTER_FILL_DATA".FILL_STATION_5[5].FILL_SEQ_OUT.Filled_Dat,
                    OutxDomestic_Cylinder => "MASTER_FILL_DATA".FILL_STATION_5[5].FILL_SEQ_OUT.Domestic_Cyl,
                    OutxCommercial_Cylinder => "MASTER_FILL_DATA".FILL_STATION_5[5].FILL_SEQ_OUT.Commercial_Cyl,
                    OutxStart_Timeout => %DB505.DBX25.0,
                    OutxTare_Entry_Error => %DB505.DBX25.1,
                    Outx_Filling_Error => %DB505.DBX25.2,
                    Outx_Tare_Value_Error => %DB505.DBX25.3,
                    Cycle_Started => #FILL_SEQ_STARTED_L2[5],
                    OutiStep_No => "MASTER_FILL_DATA".FILL_STATION_5[5].FILL_SEQ_OUT.Step_No,
                    OUTxFilling_Done => #FILLING_DONE_L2[5],
                    Gross_Weight => "CylinderSetup_DB".Array_S5[5].rGross_Weight,
                    Net_Wieght => "CylinderSetup_DB".Array_S5[5].rNet_weight);
   END_IF;
END_REGION

REGION Network 8: Call Filling Line-1 Station-6 FB
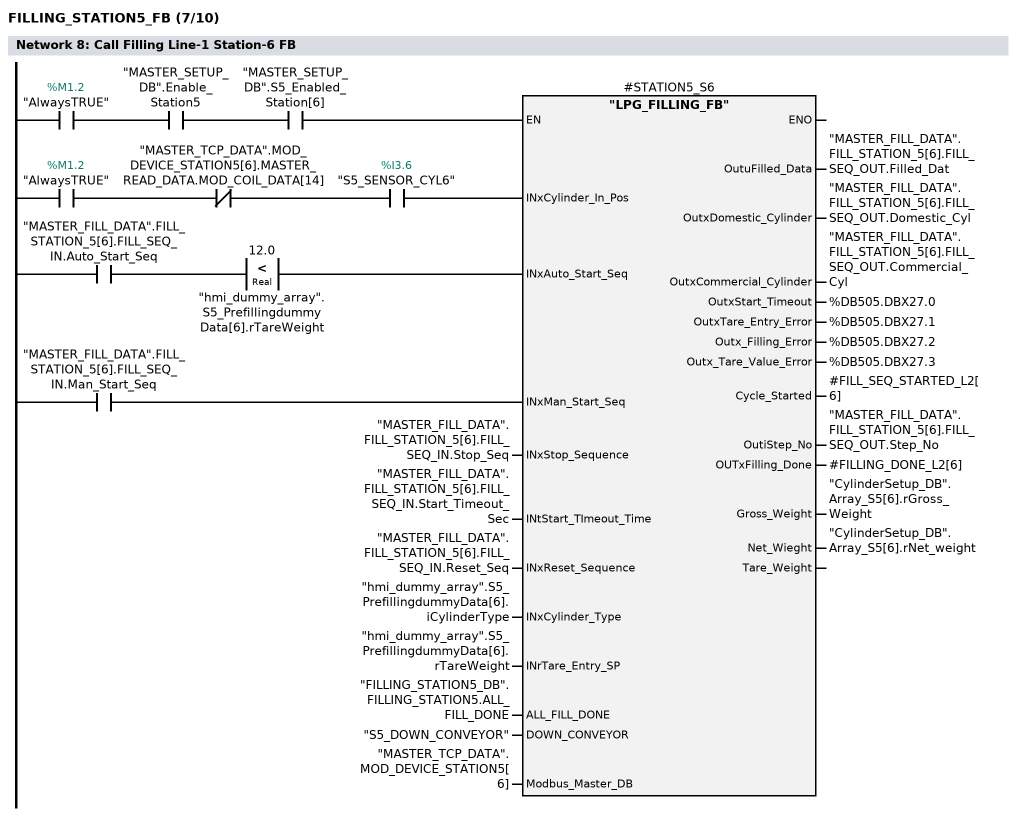
   RUNG wire#powerrail
      Contact( "AlwaysTRUE" )
      Contact( "MASTER_SETUP_DB".Enable_Station5 )
      Contact( "MASTER_SETUP_DB".S5_Enabled_Station[6] )
      #STATION5_S6(INxCylinder_In_Pos := wire#w1, INxAuto_Start_Seq := wire#w2, INxMan_Start_Seq := wire#w3, INxStop_Sequence := "MASTER_FILL_DATA".FILL_STATION_5[6].FILL_SEQ_IN.Stop_Seq, INtStart_TImeout_Time := "MASTER_FILL_DATA".FILL_STATION_5[6].FILL_SEQ_IN.Start_Timeout_Sec, INxReset_Sequence := "MASTER_FILL_DATA".FILL_STATION_5[6].FILL_SEQ_IN.Reset_Seq, INxCylinder_Type := "hmi_dummy_array".S5_PrefillingdummyData[6].iCylinderType, INrTare_Entry_SP := "hmi_dummy_array".S5_PrefillingdummyData[6].rTareWeight, ALL_FILL_DONE := "FILLING_STATION5_DB".FILLING_STATION5.ALL_FILL_DONE, DOWN_CONVEYOR := "S5_DOWN_CONVEYOR", Modbus_Master_DB := "MASTER_TCP_DATA".MOD_DEVICE_STATION5[6], OutuFilled_Data => "MASTER_FILL_DATA".FILL_STATION_5[6].FILL_SEQ_OUT.Filled_Dat, OutxDomestic_Cylinder => "MASTER_FILL_DATA".FILL_STATION_5[6].FILL_SEQ_OUT.Domestic_Cyl, OutxCommercial_Cylinder => "MASTER_FILL_DATA".FILL_STATION_5[6].FILL_SEQ_OUT.Commercial_Cyl, OutxStart_Timeout => %DB505.DBX27.0, OutxTare_Entry_Error => %DB505.DBX27.1, Outx_Filling_Error => %DB505.DBX27.2, Outx_Tare_Value_Error => %DB505.DBX27.3, Cycle_Started => #FILL_SEQ_STARTED_L2[6], OutiStep_No => "MASTER_FILL_DATA".FILL_STATION_5[6].FILL_SEQ_OUT.Step_No, OUTxFilling_Done => #FILLING_DONE_L2[6], Gross_Weight => "CylinderSetup_DB".Array_S5[6].rGross_Weight, Net_Wieght => "CylinderSetup_DB".Array_S5[6].rNet_weight, Tare_Weight =>)
   END_RUNG
   RUNG wire#powerrail
      Contact( "AlwaysTRUE" )
      I_Contact( "MASTER_TCP_DATA".MOD_DEVICE_STATION5[6].MASTER_READ_DATA.MOD_COIL_DATA[14] )
      Contact( "S5_SENSOR_CYL6" )
   END_RUNG wire#w1
   RUNG wire#powerrail
      Contact( "MASTER_FILL_DATA".FILL_STATION_5[6].FILL_SEQ_IN.Auto_Start_Seq )
      { S7_Templates := "SrcType := Real" } LT_Contact(in1 := 12.0, in2 := "hmi_dummy_array".S5_PrefillingdummyData[6].rTareWeight)
   END_RUNG wire#w2
   RUNG wire#powerrail
      Contact( "MASTER_FILL_DATA".FILL_STATION_5[6].FILL_SEQ_IN.Man_Start_Seq )
   END_RUNG wire#w3
   // the same network as SCL:
   IF "AlwaysTRUE" AND "MASTER_SETUP_DB".Enable_Station5 AND "MASTER_SETUP_DB".S5_Enabled_Station[6] THEN
       #STATION5_S6(INxCylinder_In_Pos := "AlwaysTRUE" AND NOT "MASTER_TCP_DATA".MOD_DEVICE_STATION5[6].MASTER_READ_DATA.MOD_COIL_DATA[14] AND "S5_SENSOR_CYL6",   // "LPG_FILLING_FB"
                    INxAuto_Start_Seq := "MASTER_FILL_DATA".FILL_STATION_5[6].FILL_SEQ_IN.Auto_Start_Seq AND (12.0 < "hmi_dummy_array".S5_PrefillingdummyData[6].rTareWeight),
                    INxMan_Start_Seq := "MASTER_FILL_DATA".FILL_STATION_5[6].FILL_SEQ_IN.Man_Start_Seq,
                    INxStop_Sequence := "MASTER_FILL_DATA".FILL_STATION_5[6].FILL_SEQ_IN.Stop_Seq,
                    INtStart_TImeout_Time := "MASTER_FILL_DATA".FILL_STATION_5[6].FILL_SEQ_IN.Start_Timeout_Sec,
                    INxReset_Sequence := "MASTER_FILL_DATA".FILL_STATION_5[6].FILL_SEQ_IN.Reset_Seq,
                    INxCylinder_Type := "hmi_dummy_array".S5_PrefillingdummyData[6].iCylinderType,
                    INrTare_Entry_SP := "hmi_dummy_array".S5_PrefillingdummyData[6].rTareWeight,
                    ALL_FILL_DONE := "FILLING_STATION5_DB".FILLING_STATION5.ALL_FILL_DONE,
                    DOWN_CONVEYOR := "S5_DOWN_CONVEYOR",
                    Modbus_Master_DB := "MASTER_TCP_DATA".MOD_DEVICE_STATION5[6],
                    OutuFilled_Data => "MASTER_FILL_DATA".FILL_STATION_5[6].FILL_SEQ_OUT.Filled_Dat,
                    OutxDomestic_Cylinder => "MASTER_FILL_DATA".FILL_STATION_5[6].FILL_SEQ_OUT.Domestic_Cyl,
                    OutxCommercial_Cylinder => "MASTER_FILL_DATA".FILL_STATION_5[6].FILL_SEQ_OUT.Commercial_Cyl,
                    OutxStart_Timeout => %DB505.DBX27.0,
                    OutxTare_Entry_Error => %DB505.DBX27.1,
                    Outx_Filling_Error => %DB505.DBX27.2,
                    Outx_Tare_Value_Error => %DB505.DBX27.3,
                    Cycle_Started => #FILL_SEQ_STARTED_L2[6],
                    OutiStep_No => "MASTER_FILL_DATA".FILL_STATION_5[6].FILL_SEQ_OUT.Step_No,
                    OUTxFilling_Done => #FILLING_DONE_L2[6],
                    Gross_Weight => "CylinderSetup_DB".Array_S5[6].rGross_Weight,
                    Net_Wieght => "CylinderSetup_DB".Array_S5[6].rNet_weight);
   END_IF;
END_REGION

REGION Network 9: Reset Sequence
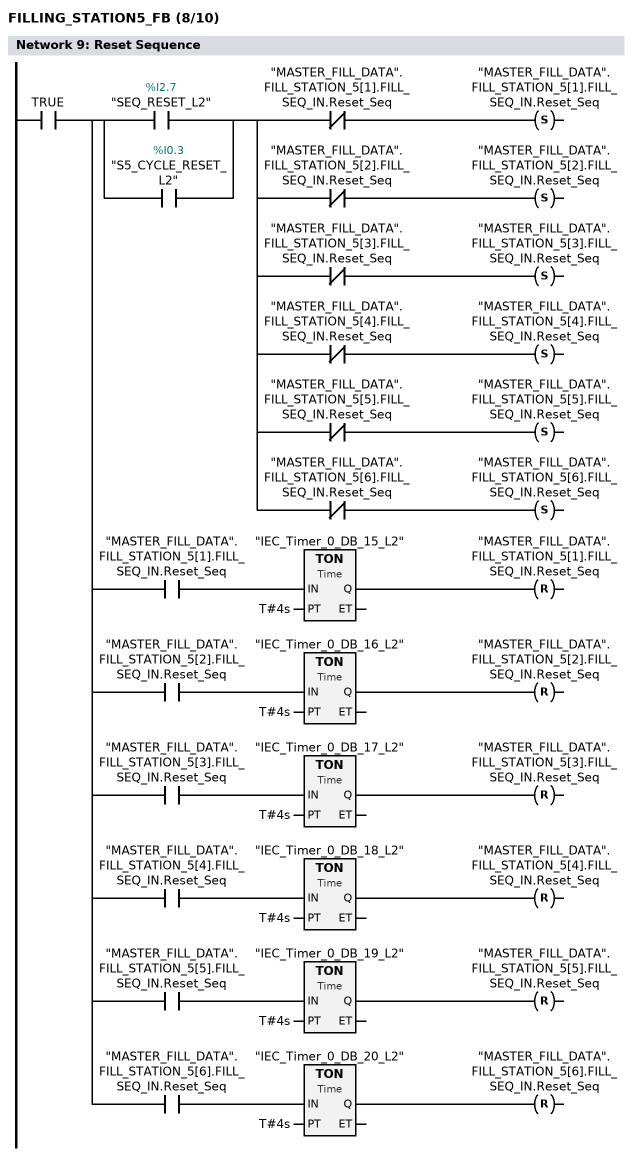
   RUNG wire#powerrail
      Contact( TRUE )
      wire#w1
      Contact( "SEQ_RESET_L2" )
      wire#w2
      I_Contact( "MASTER_FILL_DATA".FILL_STATION_5[1].FILL_SEQ_IN.Reset_Seq )
      S_Coil( "MASTER_FILL_DATA".FILL_STATION_5[1].FILL_SEQ_IN.Reset_Seq )
   END_RUNG
   RUNG wire#w1
      Contact( "S5_CYCLE_RESET_L2" )
   END_RUNG wire#w2
   RUNG wire#w2
      I_Contact( "MASTER_FILL_DATA".FILL_STATION_5[2].FILL_SEQ_IN.Reset_Seq )
      S_Coil( "MASTER_FILL_DATA".FILL_STATION_5[2].FILL_SEQ_IN.Reset_Seq )
   END_RUNG
   RUNG wire#w2
      I_Contact( "MASTER_FILL_DATA".FILL_STATION_5[3].FILL_SEQ_IN.Reset_Seq )
      S_Coil( "MASTER_FILL_DATA".FILL_STATION_5[3].FILL_SEQ_IN.Reset_Seq )
   END_RUNG
   RUNG wire#w2
      I_Contact( "MASTER_FILL_DATA".FILL_STATION_5[4].FILL_SEQ_IN.Reset_Seq )
      S_Coil( "MASTER_FILL_DATA".FILL_STATION_5[4].FILL_SEQ_IN.Reset_Seq )
   END_RUNG
   RUNG wire#w2
      I_Contact( "MASTER_FILL_DATA".FILL_STATION_5[5].FILL_SEQ_IN.Reset_Seq )
      S_Coil( "MASTER_FILL_DATA".FILL_STATION_5[5].FILL_SEQ_IN.Reset_Seq )
   END_RUNG
   RUNG wire#w2
      I_Contact( "MASTER_FILL_DATA".FILL_STATION_5[6].FILL_SEQ_IN.Reset_Seq )
      S_Coil( "MASTER_FILL_DATA".FILL_STATION_5[6].FILL_SEQ_IN.Reset_Seq )
   END_RUNG
   RUNG wire#w1
      Contact( "MASTER_FILL_DATA".FILL_STATION_5[1].FILL_SEQ_IN.Reset_Seq )
      { S7_Templates := "time_type := Time" } "IEC_Timer_0_DB_15_L2".TON(pt := T#4s, et =>)
      R_Coil( "MASTER_FILL_DATA".FILL_STATION_5[1].FILL_SEQ_IN.Reset_Seq )
   END_RUNG
   RUNG wire#w1
      Contact( "MASTER_FILL_DATA".FILL_STATION_5[2].FILL_SEQ_IN.Reset_Seq )
      { S7_Templates := "time_type := Time" } "IEC_Timer_0_DB_16_L2".TON(pt := T#4s, et =>)
      R_Coil( "MASTER_FILL_DATA".FILL_STATION_5[2].FILL_SEQ_IN.Reset_Seq )
   END_RUNG
   RUNG wire#w1
      Contact( "MASTER_FILL_DATA".FILL_STATION_5[3].FILL_SEQ_IN.Reset_Seq )
      { S7_Templates := "time_type := Time" } "IEC_Timer_0_DB_17_L2".TON(pt := T#4s, et =>)
      R_Coil( "MASTER_FILL_DATA".FILL_STATION_5[3].FILL_SEQ_IN.Reset_Seq )
   END_RUNG
   RUNG wire#w1
      Contact( "MASTER_FILL_DATA".FILL_STATION_5[4].FILL_SEQ_IN.Reset_Seq )
      { S7_Templates := "time_type := Time" } "IEC_Timer_0_DB_18_L2".TON(pt := T#4s, et =>)
      R_Coil( "MASTER_FILL_DATA".FILL_STATION_5[4].FILL_SEQ_IN.Reset_Seq )
   END_RUNG
   RUNG wire#w1
      Contact( "MASTER_FILL_DATA".FILL_STATION_5[5].FILL_SEQ_IN.Reset_Seq )
      { S7_Templates := "time_type := Time" } "IEC_Timer_0_DB_19_L2".TON(pt := T#4s, et =>)
      R_Coil( "MASTER_FILL_DATA".FILL_STATION_5[5].FILL_SEQ_IN.Reset_Seq )
   END_RUNG
   RUNG wire#w1
      Contact( "MASTER_FILL_DATA".FILL_STATION_5[6].FILL_SEQ_IN.Reset_Seq )
      { S7_Templates := "time_type := Time" } "IEC_Timer_0_DB_20_L2".TON(pt := T#4s, et =>)
      R_Coil( "MASTER_FILL_DATA".FILL_STATION_5[6].FILL_SEQ_IN.Reset_Seq )
   END_RUNG
   // the same network as SCL:
   #_w1 := TRUE AND ("SEQ_RESET_L2" OR "S5_CYCLE_RESET_L2");
   IF #_w1 AND NOT "MASTER_FILL_DATA".FILL_STATION_5[1].FILL_SEQ_IN.Reset_Seq THEN
       "MASTER_FILL_DATA".FILL_STATION_5[1].FILL_SEQ_IN.Reset_Seq := TRUE;
   END_IF;
   IF #_w1 AND NOT "MASTER_FILL_DATA".FILL_STATION_5[2].FILL_SEQ_IN.Reset_Seq THEN
       "MASTER_FILL_DATA".FILL_STATION_5[2].FILL_SEQ_IN.Reset_Seq := TRUE;
   END_IF;
   IF #_w1 AND NOT "MASTER_FILL_DATA".FILL_STATION_5[3].FILL_SEQ_IN.Reset_Seq THEN
       "MASTER_FILL_DATA".FILL_STATION_5[3].FILL_SEQ_IN.Reset_Seq := TRUE;
   END_IF;
   IF #_w1 AND NOT "MASTER_FILL_DATA".FILL_STATION_5[4].FILL_SEQ_IN.Reset_Seq THEN
       "MASTER_FILL_DATA".FILL_STATION_5[4].FILL_SEQ_IN.Reset_Seq := TRUE;
   END_IF;
   IF #_w1 AND NOT "MASTER_FILL_DATA".FILL_STATION_5[5].FILL_SEQ_IN.Reset_Seq THEN
       "MASTER_FILL_DATA".FILL_STATION_5[5].FILL_SEQ_IN.Reset_Seq := TRUE;
   END_IF;
   IF #_w1 AND NOT "MASTER_FILL_DATA".FILL_STATION_5[6].FILL_SEQ_IN.Reset_Seq THEN
       "MASTER_FILL_DATA".FILL_STATION_5[6].FILL_SEQ_IN.Reset_Seq := TRUE;
   END_IF;
   "IEC_Timer_0_DB_15_L2".TON(IN := TRUE AND "MASTER_FILL_DATA".FILL_STATION_5[1].FILL_SEQ_IN.Reset_Seq,
                           PT := T#4s);
   IF "IEC_Timer_0_DB_15_L2".Q THEN
       "MASTER_FILL_DATA".FILL_STATION_5[1].FILL_SEQ_IN.Reset_Seq := FALSE;
   END_IF;
   "IEC_Timer_0_DB_16_L2".TON(IN := TRUE AND "MASTER_FILL_DATA".FILL_STATION_5[2].FILL_SEQ_IN.Reset_Seq,
                           PT := T#4s);
   IF "IEC_Timer_0_DB_16_L2".Q THEN
       "MASTER_FILL_DATA".FILL_STATION_5[2].FILL_SEQ_IN.Reset_Seq := FALSE;
   END_IF;
   "IEC_Timer_0_DB_17_L2".TON(IN := TRUE AND "MASTER_FILL_DATA".FILL_STATION_5[3].FILL_SEQ_IN.Reset_Seq,
                           PT := T#4s);
   IF "IEC_Timer_0_DB_17_L2".Q THEN
       "MASTER_FILL_DATA".FILL_STATION_5[3].FILL_SEQ_IN.Reset_Seq := FALSE;
   END_IF;
   "IEC_Timer_0_DB_18_L2".TON(IN := TRUE AND "MASTER_FILL_DATA".FILL_STATION_5[4].FILL_SEQ_IN.Reset_Seq,
                           PT := T#4s);
   IF "IEC_Timer_0_DB_18_L2".Q THEN
       "MASTER_FILL_DATA".FILL_STATION_5[4].FILL_SEQ_IN.Reset_Seq := FALSE;
   END_IF;
   "IEC_Timer_0_DB_19_L2".TON(IN := TRUE AND "MASTER_FILL_DATA".FILL_STATION_5[5].FILL_SEQ_IN.Reset_Seq,
                           PT := T#4s);
   IF "IEC_Timer_0_DB_19_L2".Q THEN
       "MASTER_FILL_DATA".FILL_STATION_5[5].FILL_SEQ_IN.Reset_Seq := FALSE;
   END_IF;
   "IEC_Timer_0_DB_20_L2".TON(IN := TRUE AND "MASTER_FILL_DATA".FILL_STATION_5[6].FILL_SEQ_IN.Reset_Seq,
                           PT := T#4s);
   IF "IEC_Timer_0_DB_20_L2".Q THEN
       "MASTER_FILL_DATA".FILL_STATION_5[6].FILL_SEQ_IN.Reset_Seq := FALSE;
   END_IF;
END_REGION

REGION Network 10: Reset Sequence
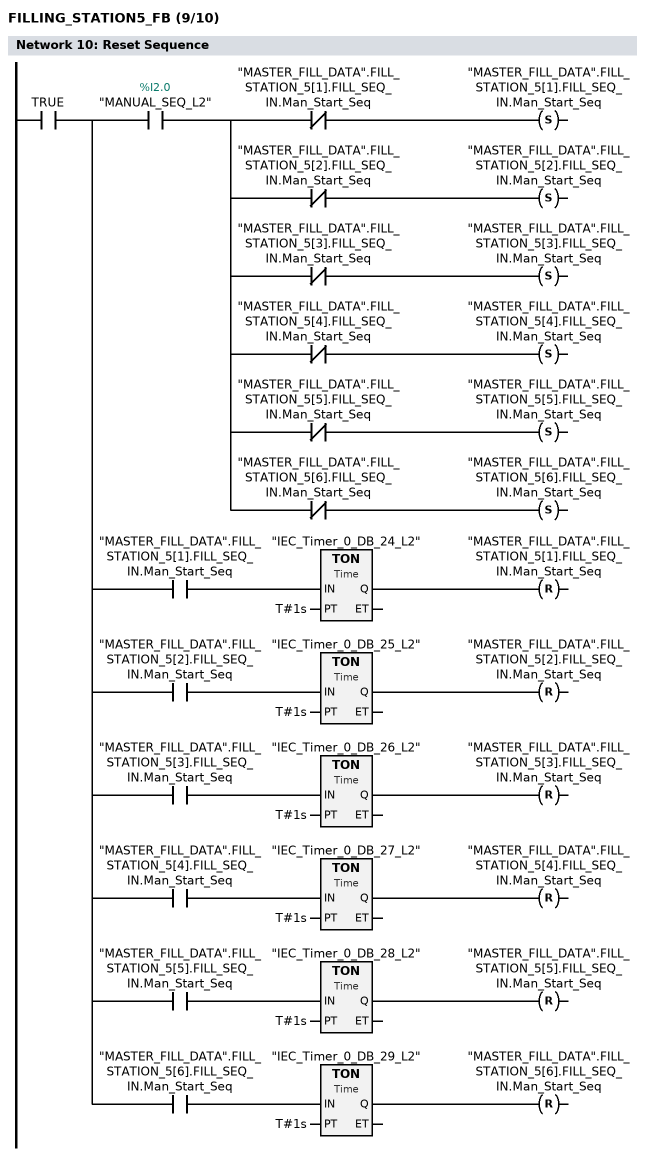
   RUNG wire#powerrail
      Contact( TRUE )
      wire#w1
      Contact( "MANUAL_SEQ_L2" )
      wire#w2
      I_Contact( "MASTER_FILL_DATA".FILL_STATION_5[1].FILL_SEQ_IN.Man_Start_Seq )
      S_Coil( "MASTER_FILL_DATA".FILL_STATION_5[1].FILL_SEQ_IN.Man_Start_Seq )
   END_RUNG
   RUNG wire#w2
      I_Contact( "MASTER_FILL_DATA".FILL_STATION_5[2].FILL_SEQ_IN.Man_Start_Seq )
      S_Coil( "MASTER_FILL_DATA".FILL_STATION_5[2].FILL_SEQ_IN.Man_Start_Seq )
   END_RUNG
   RUNG wire#w2
      I_Contact( "MASTER_FILL_DATA".FILL_STATION_5[3].FILL_SEQ_IN.Man_Start_Seq )
      S_Coil( "MASTER_FILL_DATA".FILL_STATION_5[3].FILL_SEQ_IN.Man_Start_Seq )
   END_RUNG
   RUNG wire#w2
      I_Contact( "MASTER_FILL_DATA".FILL_STATION_5[4].FILL_SEQ_IN.Man_Start_Seq )
      S_Coil( "MASTER_FILL_DATA".FILL_STATION_5[4].FILL_SEQ_IN.Man_Start_Seq )
   END_RUNG
   RUNG wire#w2
      I_Contact( "MASTER_FILL_DATA".FILL_STATION_5[5].FILL_SEQ_IN.Man_Start_Seq )
      S_Coil( "MASTER_FILL_DATA".FILL_STATION_5[5].FILL_SEQ_IN.Man_Start_Seq )
   END_RUNG
   RUNG wire#w2
      I_Contact( "MASTER_FILL_DATA".FILL_STATION_5[6].FILL_SEQ_IN.Man_Start_Seq )
      S_Coil( "MASTER_FILL_DATA".FILL_STATION_5[6].FILL_SEQ_IN.Man_Start_Seq )
   END_RUNG
   RUNG wire#w1
      Contact( "MASTER_FILL_DATA".FILL_STATION_5[1].FILL_SEQ_IN.Man_Start_Seq )
      { S7_Templates := "time_type := Time" } "IEC_Timer_0_DB_24_L2".TON(pt := T#1s, et =>)
      R_Coil( "MASTER_FILL_DATA".FILL_STATION_5[1].FILL_SEQ_IN.Man_Start_Seq )
   END_RUNG
   RUNG wire#w1
      Contact( "MASTER_FILL_DATA".FILL_STATION_5[2].FILL_SEQ_IN.Man_Start_Seq )
      { S7_Templates := "time_type := Time" } "IEC_Timer_0_DB_25_L2".TON(pt := T#1s, et =>)
      R_Coil( "MASTER_FILL_DATA".FILL_STATION_5[2].FILL_SEQ_IN.Man_Start_Seq )
   END_RUNG
   RUNG wire#w1
      Contact( "MASTER_FILL_DATA".FILL_STATION_5[3].FILL_SEQ_IN.Man_Start_Seq )
      { S7_Templates := "time_type := Time" } "IEC_Timer_0_DB_26_L2".TON(pt := T#1s, et =>)
      R_Coil( "MASTER_FILL_DATA".FILL_STATION_5[3].FILL_SEQ_IN.Man_Start_Seq )
   END_RUNG
   RUNG wire#w1
      Contact( "MASTER_FILL_DATA".FILL_STATION_5[4].FILL_SEQ_IN.Man_Start_Seq )
      { S7_Templates := "time_type := Time" } "IEC_Timer_0_DB_27_L2".TON(pt := T#1s, et =>)
      R_Coil( "MASTER_FILL_DATA".FILL_STATION_5[4].FILL_SEQ_IN.Man_Start_Seq )
   END_RUNG
   RUNG wire#w1
      Contact( "MASTER_FILL_DATA".FILL_STATION_5[5].FILL_SEQ_IN.Man_Start_Seq )
      { S7_Templates := "time_type := Time" } "IEC_Timer_0_DB_28_L2".TON(pt := T#1s, et =>)
      R_Coil( "MASTER_FILL_DATA".FILL_STATION_5[5].FILL_SEQ_IN.Man_Start_Seq )
   END_RUNG
   RUNG wire#w1
      Contact( "MASTER_FILL_DATA".FILL_STATION_5[6].FILL_SEQ_IN.Man_Start_Seq )
      { S7_Templates := "time_type := Time" } "IEC_Timer_0_DB_29_L2".TON(pt := T#1s, et =>)
      R_Coil( "MASTER_FILL_DATA".FILL_STATION_5[6].FILL_SEQ_IN.Man_Start_Seq )
   END_RUNG
   // the same network as SCL:
   #_w1 := TRUE AND "MANUAL_SEQ_L2";
   IF #_w1 AND NOT "MASTER_FILL_DATA".FILL_STATION_5[1].FILL_SEQ_IN.Man_Start_Seq THEN
       "MASTER_FILL_DATA".FILL_STATION_5[1].FILL_SEQ_IN.Man_Start_Seq := TRUE;
   END_IF;
   IF #_w1 AND NOT "MASTER_FILL_DATA".FILL_STATION_5[2].FILL_SEQ_IN.Man_Start_Seq THEN
       "MASTER_FILL_DATA".FILL_STATION_5[2].FILL_SEQ_IN.Man_Start_Seq := TRUE;
   END_IF;
   IF #_w1 AND NOT "MASTER_FILL_DATA".FILL_STATION_5[3].FILL_SEQ_IN.Man_Start_Seq THEN
       "MASTER_FILL_DATA".FILL_STATION_5[3].FILL_SEQ_IN.Man_Start_Seq := TRUE;
   END_IF;
   IF #_w1 AND NOT "MASTER_FILL_DATA".FILL_STATION_5[4].FILL_SEQ_IN.Man_Start_Seq THEN
       "MASTER_FILL_DATA".FILL_STATION_5[4].FILL_SEQ_IN.Man_Start_Seq := TRUE;
   END_IF;
   IF #_w1 AND NOT "MASTER_FILL_DATA".FILL_STATION_5[5].FILL_SEQ_IN.Man_Start_Seq THEN
       "MASTER_FILL_DATA".FILL_STATION_5[5].FILL_SEQ_IN.Man_Start_Seq := TRUE;
   END_IF;
   IF #_w1 AND NOT "MASTER_FILL_DATA".FILL_STATION_5[6].FILL_SEQ_IN.Man_Start_Seq THEN
       "MASTER_FILL_DATA".FILL_STATION_5[6].FILL_SEQ_IN.Man_Start_Seq := TRUE;
   END_IF;
   "IEC_Timer_0_DB_24_L2".TON(IN := TRUE AND "MASTER_FILL_DATA".FILL_STATION_5[1].FILL_SEQ_IN.Man_Start_Seq,
                           PT := T#1s);
   IF "IEC_Timer_0_DB_24_L2".Q THEN
       "MASTER_FILL_DATA".FILL_STATION_5[1].FILL_SEQ_IN.Man_Start_Seq := FALSE;
   END_IF;
   "IEC_Timer_0_DB_25_L2".TON(IN := TRUE AND "MASTER_FILL_DATA".FILL_STATION_5[2].FILL_SEQ_IN.Man_Start_Seq,
                           PT := T#1s);
   IF "IEC_Timer_0_DB_25_L2".Q THEN
       "MASTER_FILL_DATA".FILL_STATION_5[2].FILL_SEQ_IN.Man_Start_Seq := FALSE;
   END_IF;
   "IEC_Timer_0_DB_26_L2".TON(IN := TRUE AND "MASTER_FILL_DATA".FILL_STATION_5[3].FILL_SEQ_IN.Man_Start_Seq,
                           PT := T#1s);
   IF "IEC_Timer_0_DB_26_L2".Q THEN
       "MASTER_FILL_DATA".FILL_STATION_5[3].FILL_SEQ_IN.Man_Start_Seq := FALSE;
   END_IF;
   "IEC_Timer_0_DB_27_L2".TON(IN := TRUE AND "MASTER_FILL_DATA".FILL_STATION_5[4].FILL_SEQ_IN.Man_Start_Seq,
                           PT := T#1s);
   IF "IEC_Timer_0_DB_27_L2".Q THEN
       "MASTER_FILL_DATA".FILL_STATION_5[4].FILL_SEQ_IN.Man_Start_Seq := FALSE;
   END_IF;
   "IEC_Timer_0_DB_28_L2".TON(IN := TRUE AND "MASTER_FILL_DATA".FILL_STATION_5[5].FILL_SEQ_IN.Man_Start_Seq,
                           PT := T#1s);
   IF "IEC_Timer_0_DB_28_L2".Q THEN
       "MASTER_FILL_DATA".FILL_STATION_5[5].FILL_SEQ_IN.Man_Start_Seq := FALSE;
   END_IF;
   "IEC_Timer_0_DB_29_L2".TON(IN := TRUE AND "MASTER_FILL_DATA".FILL_STATION_5[6].FILL_SEQ_IN.Man_Start_Seq,
                           PT := T#1s);
   IF "IEC_Timer_0_DB_29_L2".Q THEN
       "MASTER_FILL_DATA".FILL_STATION_5[6].FILL_SEQ_IN.Man_Start_Seq := FALSE;
   END_IF;
END_REGION

REGION Network 11
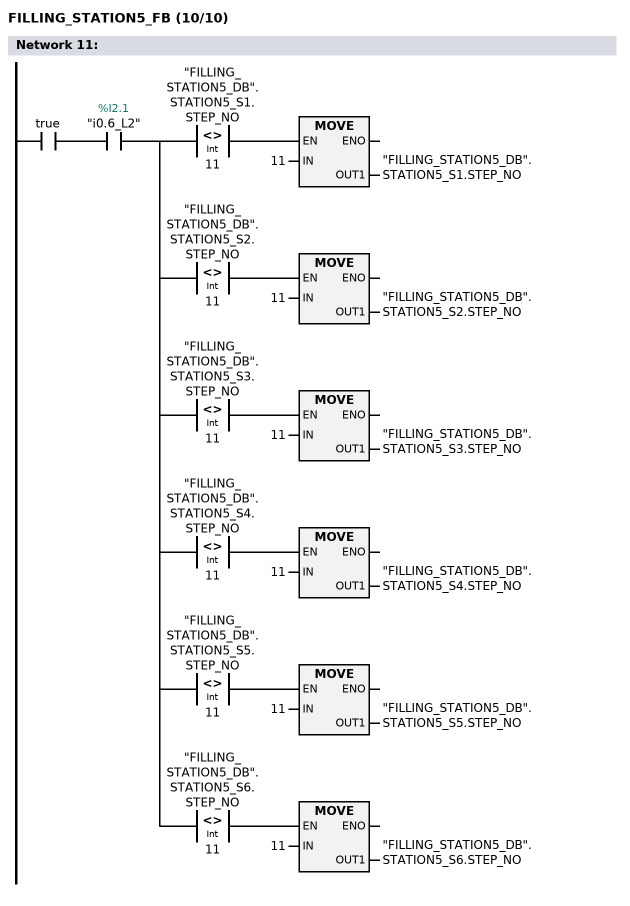
   RUNG wire#powerrail
      Contact( true )
      Contact( "i0.6_L2" )
      wire#w1
      { S7_Templates := "SrcType := Int" } NE_Contact(in1 := "FILLING_STATION5_DB".STATION5_S1.STEP_NO, in2 := 11)
      Move(in := 11, out1 => "FILLING_STATION5_DB".STATION5_S1.STEP_NO)
   END_RUNG
   RUNG wire#w1
      { S7_Templates := "SrcType := Int" } NE_Contact(in1 := "FILLING_STATION5_DB".STATION5_S2.STEP_NO, in2 := 11)
      Move(in := 11, out1 => "FILLING_STATION5_DB".STATION5_S2.STEP_NO)
   END_RUNG
   RUNG wire#w1
      { S7_Templates := "SrcType := Int" } NE_Contact(in1 := "FILLING_STATION5_DB".STATION5_S3.STEP_NO, in2 := 11)
      Move(in := 11, out1 => "FILLING_STATION5_DB".STATION5_S3.STEP_NO)
   END_RUNG
   RUNG wire#w1
      { S7_Templates := "SrcType := Int" } NE_Contact(in1 := "FILLING_STATION5_DB".STATION5_S4.STEP_NO, in2 := 11)
      Move(in := 11, out1 => "FILLING_STATION5_DB".STATION5_S4.STEP_NO)
   END_RUNG
   RUNG wire#w1
      { S7_Templates := "SrcType := Int" } NE_Contact(in1 := "FILLING_STATION5_DB".STATION5_S5.STEP_NO, in2 := 11)
      Move(in := 11, out1 => "FILLING_STATION5_DB".STATION5_S5.STEP_NO)
   END_RUNG
   RUNG wire#w1
      { S7_Templates := "SrcType := Int" } NE_Contact(in1 := "FILLING_STATION5_DB".STATION5_S6.STEP_NO, in2 := 11)
      Move(in := 11, out1 => "FILLING_STATION5_DB".STATION5_S6.STEP_NO)
   END_RUNG
   // the same network as SCL:
   #_w1 := true AND "i0.6_L2";
   IF #_w1 AND ("FILLING_STATION5_DB".STATION5_S1.STEP_NO <> 11) THEN
       "FILLING_STATION5_DB".STATION5_S1.STEP_NO := 11;
   END_IF;
   IF #_w1 AND ("FILLING_STATION5_DB".STATION5_S2.STEP_NO <> 11) THEN
       "FILLING_STATION5_DB".STATION5_S2.STEP_NO := 11;
   END_IF;
   IF #_w1 AND ("FILLING_STATION5_DB".STATION5_S3.STEP_NO <> 11) THEN
       "FILLING_STATION5_DB".STATION5_S3.STEP_NO := 11;
   END_IF;
   IF #_w1 AND ("FILLING_STATION5_DB".STATION5_S4.STEP_NO <> 11) THEN
       "FILLING_STATION5_DB".STATION5_S4.STEP_NO := 11;
   END_IF;
   IF #_w1 AND ("FILLING_STATION5_DB".STATION5_S5.STEP_NO <> 11) THEN
       "FILLING_STATION5_DB".STATION5_S5.STEP_NO := 11;
   END_IF;
   IF #_w1 AND ("FILLING_STATION5_DB".STATION5_S6.STEP_NO <> 11) THEN
       "FILLING_STATION5_DB".STATION5_S6.STEP_NO := 11;
   END_IF;
END_REGION
END_FUNCTION_BLOCK

FUNCTION_BLOCK "FILLING_FB_L2"   // FB12, LAD
{ S7_Optimized_Access := 'TRUE' }
VERSION : 0.1
// stored: AutoNumber false, IsIECCheckEnabled false, IsRetainMemResEnabled false, MemoryReserve 100, SetENOAutomatically false, UDAEnableTagReadback false
   VAR_INPUT
      CYCLE_START : Bool;
      CYCLE_RESET : Bool;
      CYL_STOPPER : Bool;
      CYL_SENSOR1 : Bool;
      CYL_SENSOR2 : Bool;
      CYL_SENSOR3 : Bool;
      CYL_SENSOR4 : Bool;
      CYL_SENSOR5 : Bool;
      CYL_SENSOR6 : Bool;
      "DOWN CONVEYOR" : Bool;
      "SENSING TIME" : DInt;
      ENABLE_CYLINDER { ExternalAccessible := 'False'; ExternalVisible := 'False'; ExternalWritable := 'False'} : Array[1..6] of Bool;
      ENABLED_CYLINDER { ExternalAccessible := 'False'; ExternalVisible := 'False'; ExternalWritable := 'False'} : Int;
      GUN_DELAY_TIME : DInt;
      FILL_SEQ_STARTED : Array[1..6] of Bool;
      FILLING_DONE : Array[1..6] of Bool;
   END_VAR
   VAR_OUTPUT
      STOPPER : Bool;
      "LIFT TABLE1" : Bool;
      "LIFT TABLE2" : Bool;
      "LIFT TABLE3" : Bool;
      "LIFT TABLE4" : Bool;
      "LIFT TABLE5" : Bool;
      "LIFT TABLE6" : Bool;
      GUN_DOWN1 : Bool;
      GUN_DOWN2 : Bool;
      GUN_DOWN3 : Bool;
      GUN_DOWN4 : Bool;
      GUN_DOWN5 : Bool;
      GUN_DOWN6 : Bool;
      CYCLE_RUNNING : Bool;
      FILL_STT_SEQ1 : Bool;
      FILL_STT_SEQ2 : Bool;
      FILL_STT_SEQ3 : Bool;
      FILL_STT_SEQ4 : Bool;
      FILL_STT_SEQ5 : Bool;
      FILL_STT_SEQ6 : Bool;
      FILLING_SEQ_DONE : Bool;
      ALL_STATION_DISABLED : Bool;
   END_VAR
   VAR
      "FIRST SCAN BIT" : Bool;
      CYCLE_OK : Bool;
      CYCLE_RESTART : Bool;
      "COUNTER RESET" : Bool;
      FIRST_CYCLE : Bool;
      "CYL COUNT  VALUE" : Int;
      "PLUS BIT" : Array[1..50] of Bool;
      "GUN DOWN" : Bool;
   END_VAR
   VAR RETAIN
      TILLTING_TIME { S7_SetPoint := 'True'} : DInt;
      M1_DECLAMP_TIME : DInt;
      CYL_COUNTER_S1 { S7_SetPoint := 'True'} : CTU_INT;
      CYL_COUNTER_S2 { S7_SetPoint := 'True'} : CTU_INT;
      CYL_COUNTER_S3 { S7_SetPoint := 'True'} : CTU_INT;
      CYL_COUNTER_S4 { S7_SetPoint := 'True'} : CTU_INT;
      CYL_COUNTER_S5 { S7_SetPoint := 'True'} : CTU_INT;
      CYL_COUNTER_S6 { S7_SetPoint := 'True'} : CTU_INT;
      CYL_COUNTER_S11 { S7_SetPoint := 'True'} : CTU_INT;
      CYL_COUNT_CONT_S1 { S7_SetPoint := 'True'} : CTU_INT;
      CYL_COUNT_CONT_S2 { S7_SetPoint := 'True'} : CTU_INT;
      CYL_COUNT_CONT_S3 { S7_SetPoint := 'True'} : CTU_INT;
      CYL_COUNT_CONT_S4 { S7_SetPoint := 'True'} : CTU_INT;
      CYL_COUNT_CONT_S5 { S7_SetPoint := 'True'} : CTU_INT;
      CYL_COUNT_CONT_S6 { S7_SetPoint := 'True'} : CTU_INT;
      "STOPPER COUNTER" { S7_SetPoint := 'True'} : CTU_INT;
   END_VAR
   VAR
      CYL_STAB_S1 { S7_SetPoint := 'True'} : TON_TIME;
      CYL_STAB_S2 { S7_SetPoint := 'True'} : TON_TIME;
      CYL_STAB_S3 { S7_SetPoint := 'True'} : TON_TIME;
      CYL_STAB_S4 { S7_SetPoint := 'True'} : TON_TIME;
      CYL_STAB_S5 { S7_SetPoint := 'True'} : TON_TIME;
      CYL_STAB_S6 { S7_SetPoint := 'True'} : TON_TIME;
      CYCLE_RST_OFF { S7_SetPoint := 'True'} : TOF_TIME;
      CYCLE_RST_ON { S7_SetPoint := 'True'} : TON_TIME;
      DECLAMP_MUL : DInt;
      DECLAMP_ADD : DInt;
      "CYL STOPPER" : Bool;
      STOP_DLY { S7_SetPoint := 'True'} : TON_TIME;
      Disable_Stations { S7_SetPoint := 'True'} : "Disable";
      First_Cylinder : Array[1..6] of Int;
      Disab_Total_Cyl : Int;
      GUN_DOWN_FBK : Bool;
      GUN_DOWN_FBK_T { S7_SetPoint := 'True'} : TON_TIME;
      AUTO_RESTART : Bool;
      GUN_DOWN_1 { S7_SetPoint := 'True'} : TON_TIME;
      GUN_DOWN_2 { S7_SetPoint := 'True'} : TON_TIME;
      GUN_DOWN_3 { S7_SetPoint := 'True'} : TON_TIME;
      GUN_DOWN_4 { S7_SetPoint := 'True'} : TON_TIME;
      GUN_DOWN_5 { S7_SetPoint := 'True'} : TON_TIME;
      GUN_DOWN_6 { S7_SetPoint := 'True'} : TON_TIME;
      FILL_STT_1 { S7_SetPoint := 'True'} : TON_TIME;
      FILL_STT_2 { S7_SetPoint := 'True'} : TON_TIME;
      FILL_STT_3 { S7_SetPoint := 'True'} : TON_TIME;
      FILL_STT_4 { S7_SetPoint := 'True'} : TON_TIME;
      FILL_STT_5 { S7_SetPoint := 'True'} : TON_TIME;
      FILL_STT_6 { S7_SetPoint := 'True'} : TON_TIME;
      ALL_FILL_DONE : Bool;
      ALL_GUN_UP : Bool;
      AUTO_CYCLE { S7_SetPoint := 'True'} : TON_TIME;
      AUTO { S7_SetPoint := 'True'} : Bool;
      MANUAL { S7_SetPoint := 'True'} : Bool;
      Man_Gun_down_1 : Bool;
      Man_Gun_down_2 : Bool;
      Man_Gun_down_3 : Bool;
      Man_Gun_down_4 : Bool;
      Man_Gun_down_5 : Bool;
      Man_Gun_down_6 : Bool;
      Man_Lift_up_1 : Bool;
      Man_Lift_up_2 : Bool;
      Man_Lift_up_3 : Bool;
      Man_Lift_up_4 : Bool;
      Man_Lift_up_5 : Bool;
      Man_Lift_up_6 : Bool;
      trig : Array[0..50] of Bool;
      "trig count" : Array[0..10] of TON_TIME;
      delay : Time;
   END_VAR
   VAR_TEMP   // added for the SCL form of the ladder/FBD networks
      _w1 : Bool;
      _w2 : Bool;
      _w3 : Bool;
      _w4 : Bool;
      _w5 : Bool;
      _w6 : Bool;
      _w7 : Bool;
      _w8 : Bool;
      _w9 : Bool;
      _w10 : Bool;
      _w11 : Bool;
      _w12 : Bool;
      _w13 : Bool;
      _w14 : Bool;
      _w15 : Bool;
      _w16 : Bool;
      _w17 : Bool;
      _w18 : Bool;
      _w19 : Bool;
      _w20 : Bool;
      _w21 : Bool;
      _w22 : Bool;
      _w23 : Bool;
      _w24 : Bool;
      _w25 : Bool;
      _w26 : Bool;
      _w27 : Bool;
      _w28 : Bool;
      _w29 : Bool;
      _w30 : Bool;
      _w31 : Bool;
   END_VAR
BEGIN

REGION Network 2: CYCLE START / POWER RESET OFF
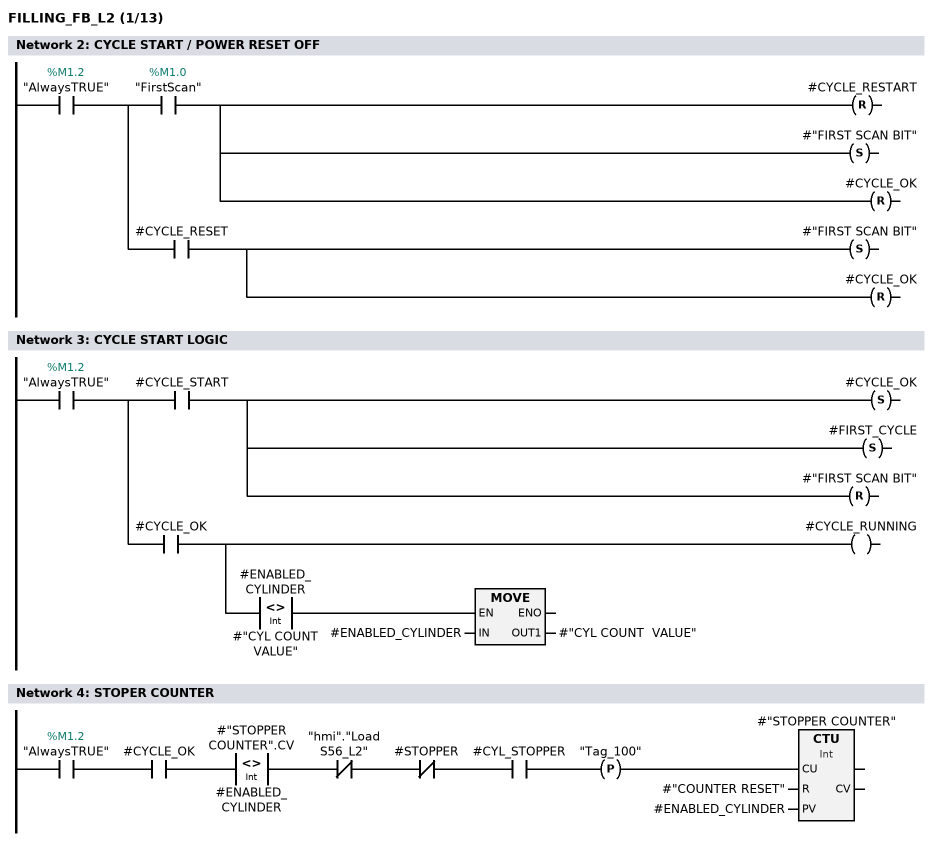
   RUNG wire#powerrail
      Contact( "AlwaysTRUE" )
      wire#w1
      Contact( "FirstScan" )
      wire#w2
      R_Coil( #CYCLE_RESTART )
   END_RUNG
   RUNG wire#w2
      S_Coil( #"FIRST SCAN BIT" )
   END_RUNG
   RUNG wire#w2
      R_Coil( #CYCLE_OK )
   END_RUNG
   RUNG wire#w1
      Contact( #CYCLE_RESET )
      wire#w3
      S_Coil( #"FIRST SCAN BIT" )
   END_RUNG
   RUNG wire#w3
      R_Coil( #CYCLE_OK )
   END_RUNG
   // the same network as SCL:
   IF "AlwaysTRUE" AND "FirstScan" THEN
       #CYCLE_RESTART := FALSE;
       #"FIRST SCAN BIT" := TRUE;
       #CYCLE_OK := FALSE;
   END_IF;
   IF "AlwaysTRUE" AND #CYCLE_RESET THEN
       #"FIRST SCAN BIT" := TRUE;
       #CYCLE_OK := FALSE;
   END_IF;
END_REGION

REGION Network 3: CYCLE START LOGIC
   RUNG wire#powerrail
      Contact( "AlwaysTRUE" )
      wire#w1
      Contact( #CYCLE_START )
      wire#w2
      S_Coil( #CYCLE_OK )
   END_RUNG
   RUNG wire#w2
      S_Coil( #FIRST_CYCLE )
   END_RUNG
   RUNG wire#w2
      R_Coil( #"FIRST SCAN BIT" )
   END_RUNG
   RUNG wire#w1
      Contact( #CYCLE_OK )
      wire#w3
      Coil( #CYCLE_RUNNING )
   END_RUNG
   RUNG wire#w3
      { S7_Templates := "SrcType := Int" } NE_Contact(in1 := #ENABLED_CYLINDER, in2 := #"CYL COUNT  VALUE")
      Move(in := #ENABLED_CYLINDER, out1 => #"CYL COUNT  VALUE")
   END_RUNG
   // the same network as SCL:
   IF "AlwaysTRUE" AND #CYCLE_START THEN
       #CYCLE_OK := TRUE;
       #FIRST_CYCLE := TRUE;
       #"FIRST SCAN BIT" := FALSE;
   END_IF;
   #CYCLE_RUNNING := "AlwaysTRUE" AND #CYCLE_OK;
   IF #CYCLE_RUNNING AND (#ENABLED_CYLINDER <> #"CYL COUNT  VALUE") THEN
       #"CYL COUNT  VALUE" := #ENABLED_CYLINDER;
   END_IF;
END_REGION

REGION Network 4: STOPER COUNTER
   RUNG wire#powerrail
      Contact( "AlwaysTRUE" )
      Contact( #CYCLE_OK )
      { S7_Templates := "SrcType := Int" } NE_Contact(in1 := #"STOPPER COUNTER".CV, in2 := #ENABLED_CYLINDER)
      I_Contact( "hmi"."Load S56_L2" )
      I_Contact( #STOPPER )
      Contact( #CYL_STOPPER )
      P_Trig( "Tag_100" )
      { S7_Templates := "value_type := Int" } #"STOPPER COUNTER".CTU(r := #"COUNTER RESET", pv := #ENABLED_CYLINDER, cv =>)
   END_RUNG
   // the same network as SCL:
   #_w1 := "AlwaysTRUE" AND #CYCLE_OK AND (#"STOPPER COUNTER".CV <> #ENABLED_CYLINDER) AND NOT "hmi"."Load S56_L2" AND NOT #STOPPER AND #CYL_STOPPER;
   #_w2 := #_w1 AND NOT "Tag_100";   // rising edge
   "Tag_100" := #_w1;
   #"STOPPER COUNTER"(CU := #_w2, R := #"COUNTER RESET", PV := #ENABLED_CYLINDER);   // CTU
END_REGION

REGION Network 5: STOPPER SET
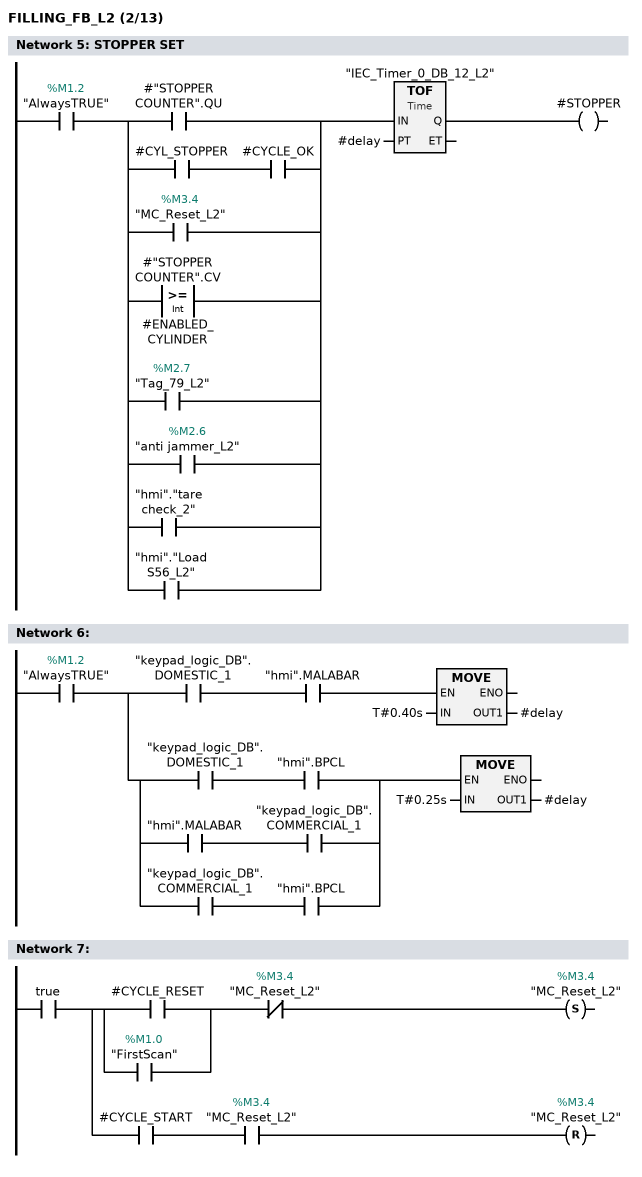
   RUNG wire#powerrail
      Contact( "AlwaysTRUE" )
      wire#w1
      Contact( #"STOPPER COUNTER".QU )
      wire#w2
      { S7_Templates := "time_type := Time" } "IEC_Timer_0_DB_12_L2".TOF(pt := #delay, et =>)
      Coil( #STOPPER )
   END_RUNG
   RUNG wire#w1
      Contact( #CYL_STOPPER )
      Contact( #CYCLE_OK )
   END_RUNG wire#w2
   RUNG wire#w1
      Contact( "MC_Reset_L2" )
   END_RUNG wire#w2
   RUNG wire#w1
      { S7_Templates := "SrcType := Int" } GE_Contact(in1 := #"STOPPER COUNTER".CV, in2 := #ENABLED_CYLINDER)
   END_RUNG wire#w2
   RUNG wire#w1
      Contact( "Tag_79_L2" )
   END_RUNG wire#w2
   RUNG wire#w1
      Contact( "anti jammer_L2" )
   END_RUNG wire#w2
   RUNG wire#w1
      Contact( "hmi"."tare check_2" )
   END_RUNG wire#w2
   RUNG wire#w1
      Contact( "hmi"."Load S56_L2" )
   END_RUNG wire#w2
   // the same network as SCL:
   "IEC_Timer_0_DB_12_L2".TOF(IN := "AlwaysTRUE" AND (#"STOPPER COUNTER".QU OR (#CYL_STOPPER AND #CYCLE_OK) OR "MC_Reset_L2" OR (#"STOPPER COUNTER".CV >= #ENABLED_CYLINDER) OR "Tag_79_L2" OR "anti jammer_L2" OR "hmi"."tare check_2" OR "hmi"."Load S56_L2"),
                           PT := #delay);
   #STOPPER := "IEC_Timer_0_DB_12_L2".Q;
END_REGION

REGION Network 6
   RUNG wire#powerrail
      Contact( "AlwaysTRUE" )
      wire#w1
      Contact( "keypad_logic_DB".DOMESTIC_1 )
      Contact( "hmi".MALABAR )
      Move(in := T#0.40s, out1 => #delay)
   END_RUNG
   RUNG wire#w1
      Contact( "keypad_logic_DB".DOMESTIC_1 )
      Contact( "hmi".BPCL )
      wire#w2
      Move(in := T#0.25s, out1 => #delay)
   END_RUNG
   RUNG wire#w1
      Contact( "hmi".MALABAR )
      Contact( "keypad_logic_DB".COMMERCIAL_1 )
   END_RUNG wire#w2
   RUNG wire#w1
      Contact( "keypad_logic_DB".COMMERCIAL_1 )
      Contact( "hmi".BPCL )
   END_RUNG wire#w2
   // the same network as SCL:
   IF "AlwaysTRUE" AND "keypad_logic_DB".DOMESTIC_1 AND "hmi".MALABAR THEN #delay := T#0.40s; END_IF;
   IF "AlwaysTRUE" AND (("keypad_logic_DB".DOMESTIC_1 AND "hmi".BPCL) OR ("hmi".MALABAR AND "keypad_logic_DB".COMMERCIAL_1) OR ("keypad_logic_DB".COMMERCIAL_1 AND "hmi".BPCL)) THEN
       #delay := T#0.25s;
   END_IF;
END_REGION

REGION Network 7
   RUNG wire#powerrail
      Contact( true )
      wire#w1
      Contact( #CYCLE_RESET )
      wire#w2
      I_Contact( "MC_Reset_L2" )
      S_Coil( "MC_Reset_L2" )
   END_RUNG
   RUNG wire#w1
      Contact( "FirstScan" )
   END_RUNG wire#w2
   RUNG wire#w1
      Contact( #CYCLE_START )
      Contact( "MC_Reset_L2" )
      R_Coil( "MC_Reset_L2" )
   END_RUNG
   // the same network as SCL:
   IF true AND (#CYCLE_RESET OR "FirstScan") AND NOT "MC_Reset_L2" THEN "MC_Reset_L2" := TRUE; END_IF;
   IF true AND #CYCLE_START AND "MC_Reset_L2" THEN "MC_Reset_L2" := FALSE; END_IF;
END_REGION

REGION Network 8: DISABLED STATIONS
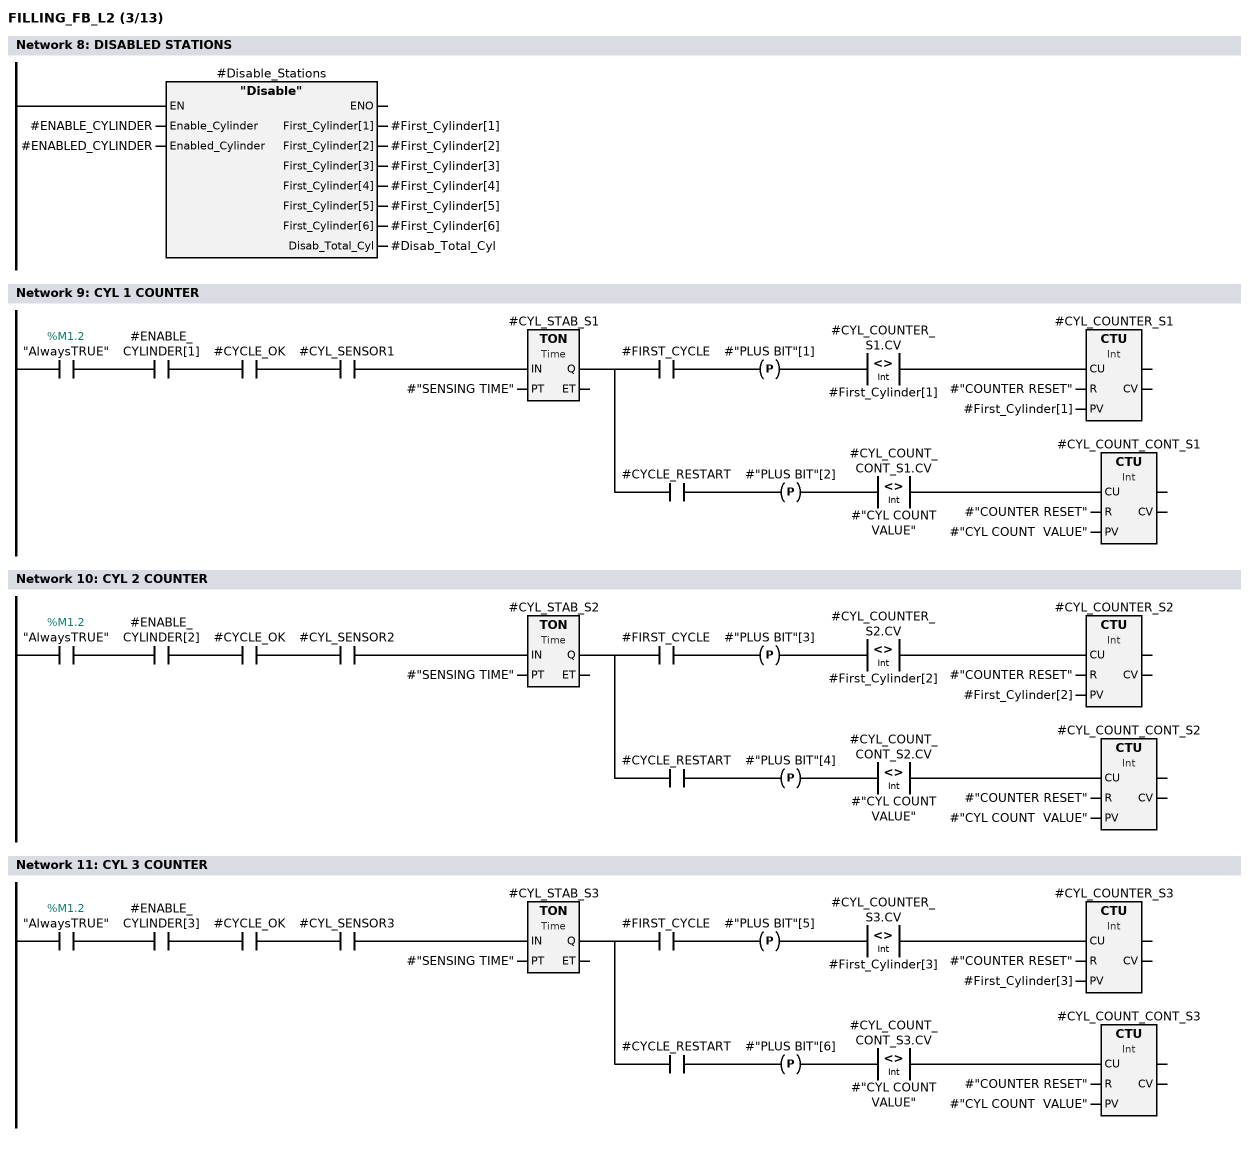
   RUNG wire#powerrail
      #Disable_Stations(Enable_Cylinder := #ENABLE_CYLINDER, Enabled_Cylinder := #ENABLED_CYLINDER, "First_Cylinder[1]" => #First_Cylinder[1], "First_Cylinder[2]" => #First_Cylinder[2], "First_Cylinder[3]" => #First_Cylinder[3], "First_Cylinder[4]" => #First_Cylinder[4], "First_Cylinder[5]" => #First_Cylinder[5], "First_Cylinder[6]" => #First_Cylinder[6], Disab_Total_Cyl => #Disab_Total_Cyl)
   END_RUNG
   // the same network as SCL:
   #Disable_Stations(Enable_Cylinder := #ENABLE_CYLINDER,   // "Disable"
                     Enabled_Cylinder := #ENABLED_CYLINDER,
                     "First_Cylinder[1]" => #First_Cylinder[1],
                     "First_Cylinder[2]" => #First_Cylinder[2],
                     "First_Cylinder[3]" => #First_Cylinder[3],
                     "First_Cylinder[4]" => #First_Cylinder[4],
                     "First_Cylinder[5]" => #First_Cylinder[5],
                     "First_Cylinder[6]" => #First_Cylinder[6],
                     Disab_Total_Cyl => #Disab_Total_Cyl);
END_REGION

REGION Network 9: CYL 1 COUNTER
   RUNG wire#powerrail
      Contact( "AlwaysTRUE" )
      Contact( #ENABLE_CYLINDER[1] )
      Contact( #CYCLE_OK )
      Contact( #CYL_SENSOR1 )
      { S7_Templates := "time_type := Time" } #CYL_STAB_S1.TON(pt := #"SENSING TIME", et =>)
      wire#w1
      Contact( #FIRST_CYCLE )
      P_Trig( #"PLUS BIT"[1] )
      { S7_Templates := "SrcType := Int" } NE_Contact(in1 := #CYL_COUNTER_S1.CV, in2 := #First_Cylinder[1])
      { S7_Templates := "value_type := Int" } #CYL_COUNTER_S1.CTU(r := #"COUNTER RESET", pv := #First_Cylinder[1], cv =>)
   END_RUNG
   RUNG wire#w1
      Contact( #CYCLE_RESTART )
      P_Trig( #"PLUS BIT"[2] )
      { S7_Templates := "SrcType := Int" } NE_Contact(in1 := #CYL_COUNT_CONT_S1.CV, in2 := #"CYL COUNT  VALUE")
      { S7_Templates := "value_type := Int" } #CYL_COUNT_CONT_S1.CTU(r := #"COUNTER RESET", pv := #"CYL COUNT  VALUE", cv =>)
   END_RUNG
   // the same network as SCL:
   #CYL_STAB_S1(IN := "AlwaysTRUE" AND #ENABLE_CYLINDER[1] AND #CYCLE_OK AND #CYL_SENSOR1,   // TON
                PT := #"SENSING TIME");
   #_w1 := #CYL_STAB_S1.Q AND #FIRST_CYCLE;
   #_w2 := #_w1 AND NOT #"PLUS BIT"[1];   // rising edge
   #"PLUS BIT"[1] := #_w1;
   #CYL_COUNTER_S1(CU := #_w2 AND (#CYL_COUNTER_S1.CV <> #First_Cylinder[1]),   // CTU
                   R := #"COUNTER RESET",
                   PV := #First_Cylinder[1]);
   #_w3 := #CYL_STAB_S1.Q AND #CYCLE_RESTART;
   #_w4 := #_w3 AND NOT #"PLUS BIT"[2];   // rising edge
   #"PLUS BIT"[2] := #_w3;
   #CYL_COUNT_CONT_S1(CU := #_w4 AND (#CYL_COUNT_CONT_S1.CV <> #"CYL COUNT  VALUE"),   // CTU
                      R := #"COUNTER RESET",
                      PV := #"CYL COUNT  VALUE");
END_REGION

REGION Network 10: CYL 2 COUNTER
   RUNG wire#powerrail
      Contact( "AlwaysTRUE" )
      Contact( #ENABLE_CYLINDER[2] )
      Contact( #CYCLE_OK )
      Contact( #CYL_SENSOR2 )
      { S7_Templates := "time_type := Time" } #CYL_STAB_S2.TON(pt := #"SENSING TIME", et =>)
      wire#w1
      Contact( #FIRST_CYCLE )
      P_Trig( #"PLUS BIT"[3] )
      { S7_Templates := "SrcType := Int" } NE_Contact(in1 := #CYL_COUNTER_S2.CV, in2 := #First_Cylinder[2])
      { S7_Templates := "value_type := Int" } #CYL_COUNTER_S2.CTU(r := #"COUNTER RESET", pv := #First_Cylinder[2], cv =>)
   END_RUNG
   RUNG wire#w1
      Contact( #CYCLE_RESTART )
      P_Trig( #"PLUS BIT"[4] )
      { S7_Templates := "SrcType := Int" } NE_Contact(in1 := #CYL_COUNT_CONT_S2.CV, in2 := #"CYL COUNT  VALUE")
      { S7_Templates := "value_type := Int" } #CYL_COUNT_CONT_S2.CTU(r := #"COUNTER RESET", pv := #"CYL COUNT  VALUE", cv =>)
   END_RUNG
   // the same network as SCL:
   #CYL_STAB_S2(IN := "AlwaysTRUE" AND #ENABLE_CYLINDER[2] AND #CYCLE_OK AND #CYL_SENSOR2,   // TON
                PT := #"SENSING TIME");
   #_w1 := #CYL_STAB_S2.Q AND #FIRST_CYCLE;
   #_w2 := #_w1 AND NOT #"PLUS BIT"[3];   // rising edge
   #"PLUS BIT"[3] := #_w1;
   #CYL_COUNTER_S2(CU := #_w2 AND (#CYL_COUNTER_S2.CV <> #First_Cylinder[2]),   // CTU
                   R := #"COUNTER RESET",
                   PV := #First_Cylinder[2]);
   #_w3 := #CYL_STAB_S2.Q AND #CYCLE_RESTART;
   #_w4 := #_w3 AND NOT #"PLUS BIT"[4];   // rising edge
   #"PLUS BIT"[4] := #_w3;
   #CYL_COUNT_CONT_S2(CU := #_w4 AND (#CYL_COUNT_CONT_S2.CV <> #"CYL COUNT  VALUE"),   // CTU
                      R := #"COUNTER RESET",
                      PV := #"CYL COUNT  VALUE");
END_REGION

REGION Network 11: CYL 3 COUNTER
   RUNG wire#powerrail
      Contact( "AlwaysTRUE" )
      Contact( #ENABLE_CYLINDER[3] )
      Contact( #CYCLE_OK )
      Contact( #CYL_SENSOR3 )
      { S7_Templates := "time_type := Time" } #CYL_STAB_S3.TON(pt := #"SENSING TIME", et =>)
      wire#w1
      Contact( #FIRST_CYCLE )
      P_Trig( #"PLUS BIT"[5] )
      { S7_Templates := "SrcType := Int" } NE_Contact(in1 := #CYL_COUNTER_S3.CV, in2 := #First_Cylinder[3])
      { S7_Templates := "value_type := Int" } #CYL_COUNTER_S3.CTU(r := #"COUNTER RESET", pv := #First_Cylinder[3], cv =>)
   END_RUNG
   RUNG wire#w1
      Contact( #CYCLE_RESTART )
      P_Trig( #"PLUS BIT"[6] )
      { S7_Templates := "SrcType := Int" } NE_Contact(in1 := #CYL_COUNT_CONT_S3.CV, in2 := #"CYL COUNT  VALUE")
      { S7_Templates := "value_type := Int" } #CYL_COUNT_CONT_S3.CTU(r := #"COUNTER RESET", pv := #"CYL COUNT  VALUE", cv =>)
   END_RUNG
   // the same network as SCL:
   #CYL_STAB_S3(IN := "AlwaysTRUE" AND #ENABLE_CYLINDER[3] AND #CYCLE_OK AND #CYL_SENSOR3,   // TON
                PT := #"SENSING TIME");
   #_w1 := #CYL_STAB_S3.Q AND #FIRST_CYCLE;
   #_w2 := #_w1 AND NOT #"PLUS BIT"[5];   // rising edge
   #"PLUS BIT"[5] := #_w1;
   #CYL_COUNTER_S3(CU := #_w2 AND (#CYL_COUNTER_S3.CV <> #First_Cylinder[3]),   // CTU
                   R := #"COUNTER RESET",
                   PV := #First_Cylinder[3]);
   #_w3 := #CYL_STAB_S3.Q AND #CYCLE_RESTART;
   #_w4 := #_w3 AND NOT #"PLUS BIT"[6];   // rising edge
   #"PLUS BIT"[6] := #_w3;
   #CYL_COUNT_CONT_S3(CU := #_w4 AND (#CYL_COUNT_CONT_S3.CV <> #"CYL COUNT  VALUE"),   // CTU
                      R := #"COUNTER RESET",
                      PV := #"CYL COUNT  VALUE");
END_REGION

REGION Network 12: CYL 4 COUNTER
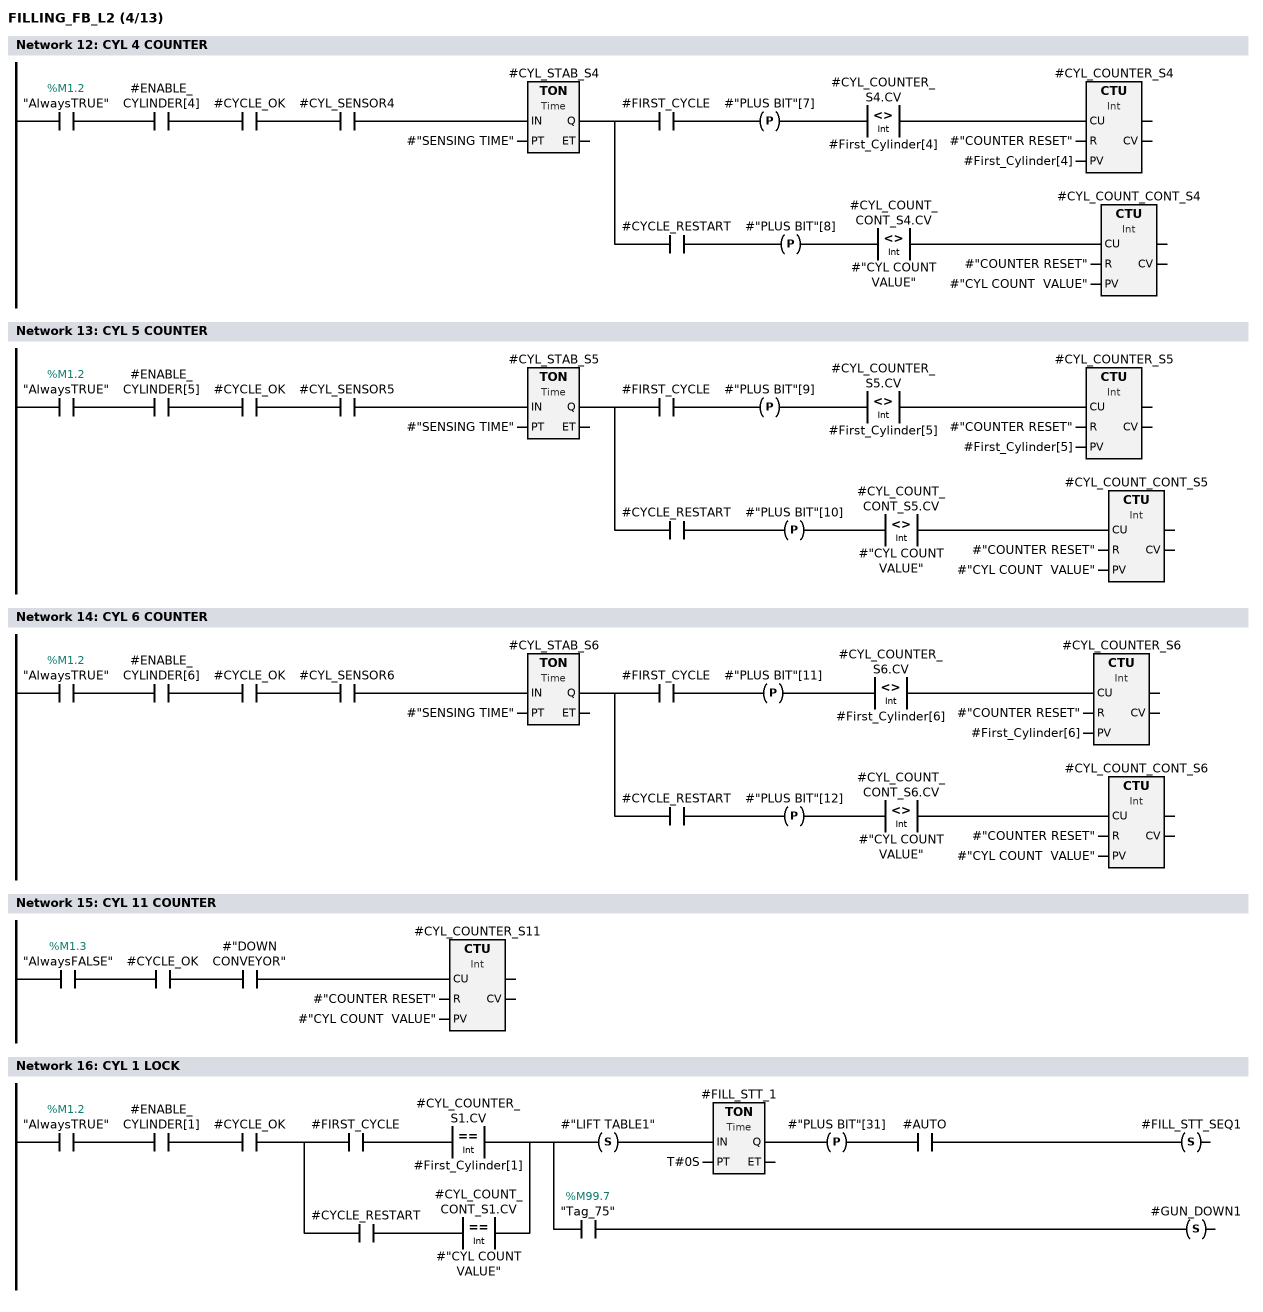
   RUNG wire#powerrail
      Contact( "AlwaysTRUE" )
      Contact( #ENABLE_CYLINDER[4] )
      Contact( #CYCLE_OK )
      Contact( #CYL_SENSOR4 )
      { S7_Templates := "time_type := Time" } #CYL_STAB_S4.TON(pt := #"SENSING TIME", et =>)
      wire#w1
      Contact( #FIRST_CYCLE )
      P_Trig( #"PLUS BIT"[7] )
      { S7_Templates := "SrcType := Int" } NE_Contact(in1 := #CYL_COUNTER_S4.CV, in2 := #First_Cylinder[4])
      { S7_Templates := "value_type := Int" } #CYL_COUNTER_S4.CTU(r := #"COUNTER RESET", pv := #First_Cylinder[4], cv =>)
   END_RUNG
   RUNG wire#w1
      Contact( #CYCLE_RESTART )
      P_Trig( #"PLUS BIT"[8] )
      { S7_Templates := "SrcType := Int" } NE_Contact(in1 := #CYL_COUNT_CONT_S4.CV, in2 := #"CYL COUNT  VALUE")
      { S7_Templates := "value_type := Int" } #CYL_COUNT_CONT_S4.CTU(r := #"COUNTER RESET", pv := #"CYL COUNT  VALUE", cv =>)
   END_RUNG
   // the same network as SCL:
   #CYL_STAB_S4(IN := "AlwaysTRUE" AND #ENABLE_CYLINDER[4] AND #CYCLE_OK AND #CYL_SENSOR4,   // TON
                PT := #"SENSING TIME");
   #_w1 := #CYL_STAB_S4.Q AND #FIRST_CYCLE;
   #_w2 := #_w1 AND NOT #"PLUS BIT"[7];   // rising edge
   #"PLUS BIT"[7] := #_w1;
   #CYL_COUNTER_S4(CU := #_w2 AND (#CYL_COUNTER_S4.CV <> #First_Cylinder[4]),   // CTU
                   R := #"COUNTER RESET",
                   PV := #First_Cylinder[4]);
   #_w3 := #CYL_STAB_S4.Q AND #CYCLE_RESTART;
   #_w4 := #_w3 AND NOT #"PLUS BIT"[8];   // rising edge
   #"PLUS BIT"[8] := #_w3;
   #CYL_COUNT_CONT_S4(CU := #_w4 AND (#CYL_COUNT_CONT_S4.CV <> #"CYL COUNT  VALUE"),   // CTU
                      R := #"COUNTER RESET",
                      PV := #"CYL COUNT  VALUE");
END_REGION

REGION Network 13: CYL 5 COUNTER
   RUNG wire#powerrail
      Contact( "AlwaysTRUE" )
      Contact( #ENABLE_CYLINDER[5] )
      Contact( #CYCLE_OK )
      Contact( #CYL_SENSOR5 )
      { S7_Templates := "time_type := Time" } #CYL_STAB_S5.TON(pt := #"SENSING TIME", et =>)
      wire#w1
      Contact( #FIRST_CYCLE )
      P_Trig( #"PLUS BIT"[9] )
      { S7_Templates := "SrcType := Int" } NE_Contact(in1 := #CYL_COUNTER_S5.CV, in2 := #First_Cylinder[5])
      { S7_Templates := "value_type := Int" } #CYL_COUNTER_S5.CTU(r := #"COUNTER RESET", pv := #First_Cylinder[5], cv =>)
   END_RUNG
   RUNG wire#w1
      Contact( #CYCLE_RESTART )
      P_Trig( #"PLUS BIT"[10] )
      { S7_Templates := "SrcType := Int" } NE_Contact(in1 := #CYL_COUNT_CONT_S5.CV, in2 := #"CYL COUNT  VALUE")
      { S7_Templates := "value_type := Int" } #CYL_COUNT_CONT_S5.CTU(r := #"COUNTER RESET", pv := #"CYL COUNT  VALUE", cv =>)
   END_RUNG
   // the same network as SCL:
   #CYL_STAB_S5(IN := "AlwaysTRUE" AND #ENABLE_CYLINDER[5] AND #CYCLE_OK AND #CYL_SENSOR5,   // TON
                PT := #"SENSING TIME");
   #_w1 := #CYL_STAB_S5.Q AND #FIRST_CYCLE;
   #_w2 := #_w1 AND NOT #"PLUS BIT"[9];   // rising edge
   #"PLUS BIT"[9] := #_w1;
   #CYL_COUNTER_S5(CU := #_w2 AND (#CYL_COUNTER_S5.CV <> #First_Cylinder[5]),   // CTU
                   R := #"COUNTER RESET",
                   PV := #First_Cylinder[5]);
   #_w3 := #CYL_STAB_S5.Q AND #CYCLE_RESTART;
   #_w4 := #_w3 AND NOT #"PLUS BIT"[10];   // rising edge
   #"PLUS BIT"[10] := #_w3;
   #CYL_COUNT_CONT_S5(CU := #_w4 AND (#CYL_COUNT_CONT_S5.CV <> #"CYL COUNT  VALUE"),   // CTU
                      R := #"COUNTER RESET",
                      PV := #"CYL COUNT  VALUE");
END_REGION

